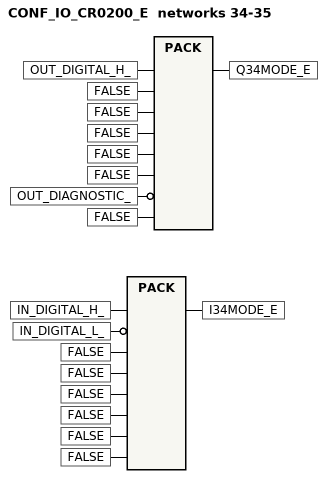
[picture p48: CONF_IO_CR0200_E (FBD) networks 34-35]
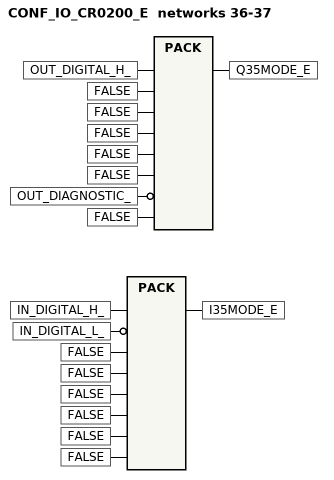
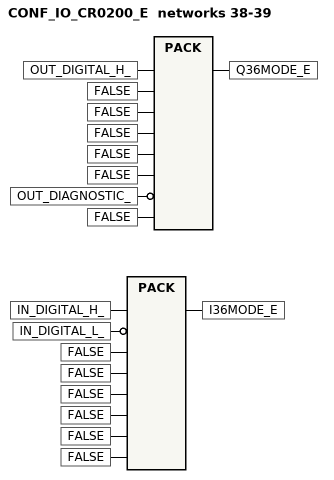
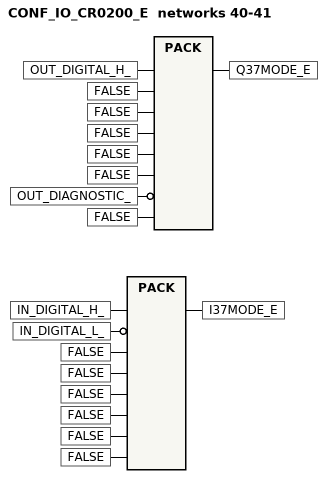
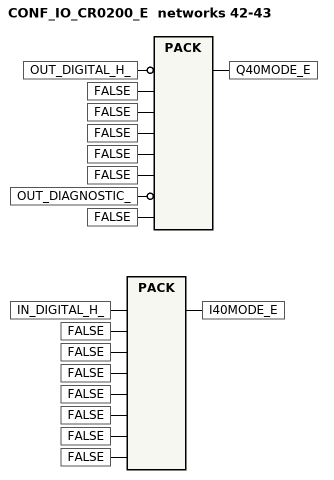
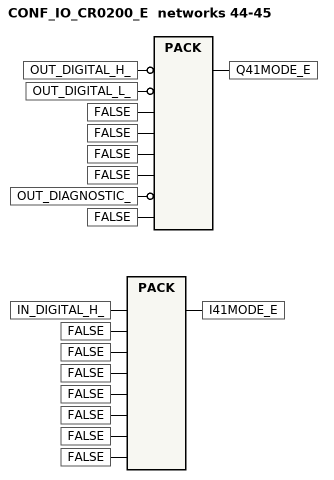
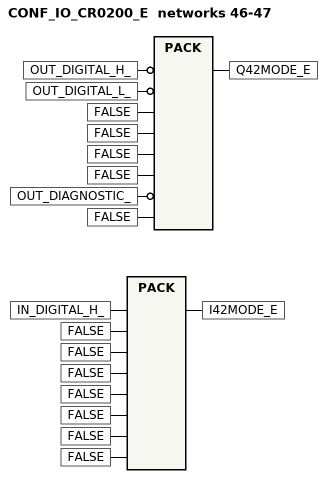
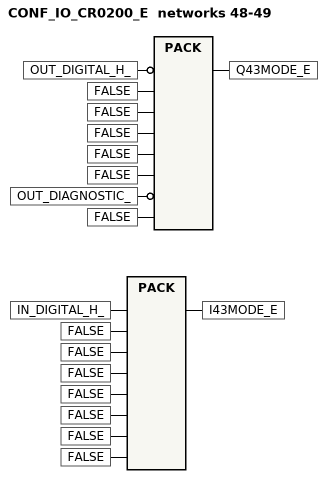
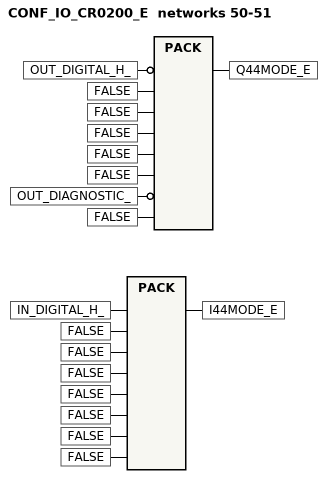
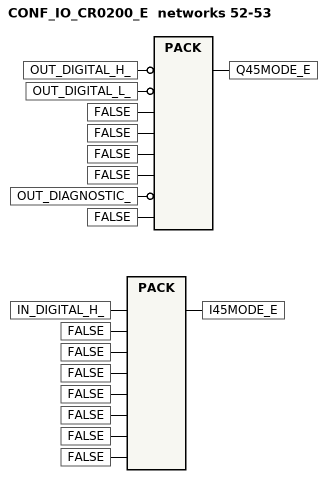
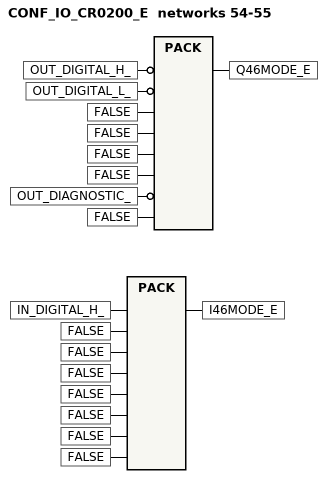
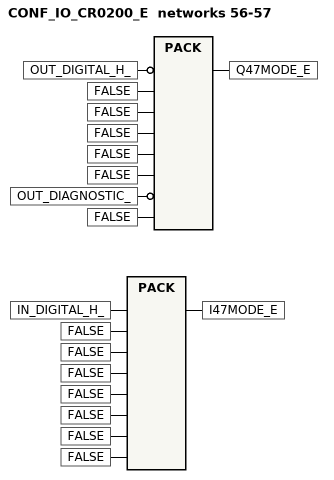
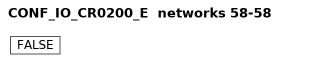
_FBD_ (* Function Block Diagram *)
NETWORK 1
	NOT init => >>END
NETWORK 2 (* Configuration byte for analog channel 0 pin 08 Connector 2. No output is connected to this pin. / Default setting:B0:=TRUE,B1:= FALSE,B2:= FALSE,B3:= FALSE,B4:= TRUE,B5:= FALSE,B6:= FALSE,B7:=FALSE *)
	PACK(IN_DIGITAL_H_, FALSE, NOT IN_CURRENT_, NOT IN_VOLTAGE10_, IN_VOLTAGE30_, NOT IN_RATIO_, FALSE, FALSE) => I00MODE_E
NETWORK 3 (* Configuration byte for analog channel 1 pin 27 Connector 2. No output is connected to this pin. / Default setting:B0:=TRUE,B1:= FALSE,B2:= FALSE,B3:= FALSE,B4:= TRUE,B5:= FALSE,B6:= FALSE,B7:=FALSE *)
	PACK(IN_DIGITAL_H_, FALSE, NOT IN_CURRENT_, NOT IN_VOLTAGE10_, IN_VOLTAGE30_, NOT IN_RATIO_, FALSE, FALSE) => I01MODE_E
NETWORK 4 (* Configuration byte for analog channel 2 pin 09 Connector 2. No output is connected to this pin. / Default setting:B0:=TRUE,B1:= FALSE,B2:= FALSE,B3:= FALSE,B4:= TRUE,B5:= FALSE,B6:= FALSE,B7:=FALSE *)
	PACK(IN_DIGITAL_H_, FALSE, NOT IN_CURRENT_, NOT IN_VOLTAGE10_, IN_VOLTAGE30_, NOT IN_RATIO_, FALSE, FALSE) => I02MODE_E
NETWORK 5 (* Configuration byte for analog channel 3 pin 28 Connector 2. No output is connected to this pin. / Default setting:B0:=TRUE,B1:= FALSE,B2:= FALSE,B3:= FALSE,B4:= TRUE,B5:= FALSE,B6:= FALSE,B7:=FALSE *)
	PACK(IN_DIGITAL_H_, FALSE, NOT IN_CURRENT_, NOT IN_VOLTAGE10_, IN_VOLTAGE30_, NOT IN_RATIO_, FALSE, FALSE) => I03MODE_E
NETWORK 6 (* Configuration byte for analog channel 4 pin 10 Connector 2. No output is connected to this pin. / Default setting:B0:=TRUE,B1:= FALSE,B2:= FALSE,B3:= FALSE,B4:= TRUE,B5:= FALSE,B6:= FALSE,B7:=FALSE *)
	PACK(IN_DIGITAL_H_, FALSE, NOT IN_CURRENT_, NOT IN_VOLTAGE10_, IN_VOLTAGE30_, NOT IN_RATIO_, FALSE, FALSE) => I04MODE_E
NETWORK 7 (* Configuration byte for analog channel 5 pin 29 Connector 2. No output is connected to this pin. / Default setting:B0:=TRUE,B1:= FALSE,B2:= FALSE,B3:= FALSE,B4:= TRUE,B5:= FALSE,B6:= FALSE,B7:=FALSE *)
	PACK(IN_DIGITAL_H_, FALSE, NOT IN_CURRENT_, NOT IN_VOLTAGE10_, IN_VOLTAGE30_, NOT IN_RATIO_, FALSE, FALSE) => I05MODE_E
NETWORK 8 (* Configuration byte for analog channel 6 pin 11 Connector 2. No output is connected to this pin. / Default setting:B0:=TRUE,B1:= FALSE,B2:= FALSE,B3:= FALSE,B4:= TRUE,B5:= FALSE,B6:= FALSE,B7:=FALSE *)
	PACK(IN_DIGITAL_H_, FALSE, NOT IN_CURRENT_, NOT IN_VOLTAGE10_, IN_VOLTAGE30_, NOT IN_RATIO_, FALSE, FALSE) => I06MODE_E
NETWORK 9 (* Configuration byte for analog channel 7 pin 30 Connector 2. No output is connected to this pin. / Default setting:B0:=TRUE,B1:= FALSE,B2:= FALSE,B3:= FALSE,B4:= TRUE,B5:= FALSE,B6:= FALSE,B7:=FALSE *)
	PACK(IN_DIGITAL_H_, FALSE, NOT IN_CURRENT_, NOT IN_VOLTAGE10_, IN_VOLTAGE30_, NOT IN_RATIO_, FALSE, FALSE) => I07MODE_E
NETWORK 10 (* Configuration byte for input %IX32.12  pin 20 Connector 2. No output is connected to this pin. / Default setting:B0:=TRUE,B1:= FALSE,B2:= FALSE,B3:= FALSE,B4:= FALSE,B5:= FALSE,B6:= FALSE,B7:=FALSE *)
	PACK(IN_DIGITAL_H_, FALSE, FALSE, FALSE, FALSE, FALSE, FALSE, NOT IN_FAST_) => I14MODE_E
NETWORK 11 (* Configuration byte for input %IX32.13  pin 02 Connector 2. No output is connected to this pin. / Default setting:B0:=TRUE,B1:= FALSE,B2:= FALSE,B3:= FALSE,B4:= FALSE,B5:= FALSE,B6:= FALSE,B7:=FALSE *)
	PACK(IN_DIGITAL_H_, FALSE, FALSE, FALSE, FALSE, FALSE, FALSE, NOT IN_FAST_) => I15MODE_E
NETWORK 12 (* Configuration byte for input %IX32.14  pin 21 Connector 2. No output is connected to this pin. / Default setting:B0:=TRUE,B1:= FALSE,B2:= FALSE,B3:= FALSE,B4:= FALSE,B5:= FALSE,B6:= FALSE,B7:=FALSE *)
	PACK(IN_DIGITAL_H_, FALSE, FALSE, FALSE, FALSE, FALSE, FALSE, NOT IN_FAST_) => I16MODE_E
NETWORK 13 (* Configuration byte for input %IX32.15  pin 38 Connector 2. No output is connected to this pin. / Default setting:B0:=TRUE,B1:= FALSE,B2:= FALSE,B3:= FALSE,B4:= FALSE,B5:= FALSE,B6:= FALSE,B7:=FALSE *)
	PACK(IN_DIGITAL_H_, FALSE, FALSE, FALSE, FALSE, FALSE, FALSE, NOT IN_FAST_) => I17MODE_E
NETWORK 14 (* Configuration byte for input %IX33.04  pin 19 Connector 2. No output is connected to this pin. / Default setting:B0:=TRUE,B1:= FALSE,B2:= FALSE,B3:= FALSE,B4:= FALSE,B5:= FALSE,B6:= FALSE,B7:=FALSE *)
	PACK(IN_DIGITAL_H_, FALSE, FALSE, FALSE, FALSE, FALSE, FALSE, NOT IN_FAST_) => I24MODE_E
NETWORK 15 (* Configuration byte for input %IX33.05  pin 55 Connector 2. No output is connected to this pin. / Default setting:B0:=TRUE,B1:= FALSE,B2:= FALSE,B3:= FALSE,B4:= FALSE,B5:= FALSE,B6:= FALSE,B7:=FALSE *)
	PACK(IN_DIGITAL_H_, FALSE, FALSE, FALSE, FALSE, FALSE, FALSE, NOT IN_FAST_) => I25MODE_E
NETWORK 16 (* Configuration byte for input %IX33.06  pin 18 Connector 2. No output is connected to this pin. / Default setting:B0:=TRUE,B1:= FALSE,B2:= FALSE,B3:= FALSE,B4:= FALSE,B5:= FALSE,B6:= FALSE,B7:=FALSE *)
	PACK(IN_DIGITAL_H_, FALSE, FALSE, FALSE, FALSE, FALSE, FALSE, NOT IN_FAST_) => I26MODE_E
NETWORK 17 (* Configuration byte for input %IX33.07  pin 37 Connector 2. No output is connected to this pin. / Default setting:B0:=TRUE,B1:= FALSE,B2:= FALSE,B3:= FALSE,B4:= FALSE,B5:= FALSE,B6:= FALSE,B7:=FALSE *)
	PACK(IN_DIGITAL_H_, FALSE, FALSE, FALSE, FALSE, FALSE, FALSE, NOT IN_FAST_) => I27MODE_E
NETWORK 18 (* Configuration byte for output %QX32.00  pin 44 Connector 2. The input %IX32.08 on pin 44 has no configuration byte. / Default setting:B0:=TRUE,B1:= FALSE,B2:= FALSE,B3:= FALSE,B4:= FALSE,B5:= FALSE,B6:= FALSE,B7:=TRUE *)
	PACK(OUT_DIGITAL_H_, FALSE, NOT OUT_CURRENT_, FALSE, FALSE, FALSE, NOT OUT_DIAGNOSTIC_, OUT_OVERLOAD_PROTECTION_) => Q10MODE_E
NETWORK 19 (* Configuration byte for output %QX32.01  pin 45 Connector 2. The input %IX32.09 on pin 45 has no configuration byte. / Default setting:B0:=TRUE,B1:= FALSE,B2:= FALSE,B3:= FALSE,B4:= FALSE,B5:= FALSE,B6:= FALSE,B7:=TRUE *)
	PACK(OUT_DIGITAL_H_, FALSE, NOT OUT_CURRENT_, FALSE, FALSE, FALSE, NOT OUT_DIAGNOSTIC_, OUT_OVERLOAD_PROTECTION_) => Q11MODE_E
NETWORK 20 (* Configuration byte for output %QX32.02  pin 46 Connector 2. The input %IX32.10 on pin 46 has no configuration byte. / Default setting:B0:=TRUE,B1:= FALSE,B2:= FALSE,B3:= FALSE,B4:= FALSE,B5:= FALSE,B6:= FALSE,B7:=TRUE *)
	PACK(OUT_DIGITAL_H_, FALSE, NOT OUT_CURRENT_, FALSE, FALSE, FALSE, NOT OUT_DIAGNOSTIC_, OUT_OVERLOAD_PROTECTION_) => Q12MODE_E
NETWORK 21 (* Configuration byte for output %QX32.03  pin 47 Connector 2. The input %IX32.11 on pin 47 has no configuration byte. / Default setting:B0:=TRUE,B1:= FALSE,B2:= FALSE,B3:= FALSE,B4:= FALSE,B5:= FALSE,B6:= FALSE,B7:=TRUE *)
	PACK(OUT_DIGITAL_H_, FALSE, NOT OUT_CURRENT_, FALSE, FALSE, FALSE, NOT OUT_DIAGNOSTIC_, OUT_OVERLOAD_PROTECTION_) => Q13MODE_E
NETWORK 22 (* Configuration byte for output %QX32.04  pin 36 Connector 2. The input %IX33.00 on pin 36 has no configuration byte. / Default setting:B0:=TRUE,B1:= FALSE,B2:= FALSE,B3:= FALSE,B4:= FALSE,B5:= FALSE,B6:= FALSE,B7:=TRUE *)
	PACK(OUT_DIGITAL_H_, FALSE, NOT OUT_CURRENT_, FALSE, FALSE, FALSE, NOT OUT_DIAGNOSTIC_, OUT_OVERLOAD_PROTECTION_) => Q20MODE_E
NETWORK 23 (* Configuration byte for output %QX32.05  pin 54 Connector 2 The input %IX33.01 on pin 54 has no configuration byte. / Default setting:B0:=TRUE,B1:= FALSE,B2:= FALSE,B3:= FALSE,B4:= FALSE,B5:= FALSE,B6:= FALSE,B7:=TRUE *)
	PACK(OUT_DIGITAL_H_, FALSE, NOT OUT_CURRENT_, FALSE, FALSE, FALSE, NOT OUT_DIAGNOSTIC_, OUT_OVERLOAD_PROTECTION_) => Q21MODE_E
NETWORK 24 (* Configuration byte for output %QX32.06  pin 17 Connector 2 The input %IX33.02 on pin 17 has no configuration byte. / Default setting:B0:=TRUE,B1:= FALSE,B2:= FALSE,B3:= FALSE,B4:= FALSE,B5:= FALSE,B6:= FALSE,B7:=TRUE *)
	PACK(OUT_DIGITAL_H_, FALSE, NOT OUT_CURRENT_, FALSE, FALSE, FALSE, NOT OUT_DIAGNOSTIC_, OUT_OVERLOAD_PROTECTION_) => Q22MODE_E
NETWORK 25 (* Configuration byte for output %QX32.07  pin 53 Connector 2 The input %IX33.03 on pin 53 has no configuration byte. / Default setting:B0:=TRUE,B1:= FALSE,B2:= FALSE,B3:= FALSE,B4:= FALSE,B5:= FALSE,B6:= FALSE,B7:=TRUE *)
	PACK(OUT_DIGITAL_H_, FALSE, NOT OUT_CURRENT_, FALSE, FALSE, FALSE, NOT OUT_DIAGNOSTIC_, OUT_OVERLOAD_PROTECTION_) => Q23MODE_E
NETWORK 26 (* Configuration byte for output %QX32.08  pin 39 Connector 2. / Default setting:B0:=TRUE,B1:= FALSE,B2:= FALSE,B3:= FALSE,B4:= FALSE,B5:= FALSE,B6:= FALSE,B7:=FALSE *)
	PACK(OUT_DIGITAL_H_, FALSE, FALSE, FALSE, FALSE, FALSE, NOT OUT_DIAGNOSTIC_, FALSE) => Q30MODE_E
NETWORK 27 (* Configuration byte for input %IX33.08  pin 39 Connector 2. / Default setting:B0:=TRUE,B1:= FALSE,B2:= FALSE,B3:= FALSE,B4:= FALSE,B5:= FALSE,B6:= FALSE,B7:=FALSE *)
	PACK(IN_DIGITAL_H_, NOT IN_DIGITAL_L_, FALSE, FALSE, FALSE, FALSE, FALSE, FALSE) => I30MODE_E
NETWORK 28 (* Configuration byte for output %QX32.09  pin 03 Connector 2. / Default setting:B0:=TRUE,B1:= FALSE,B2:= FALSE,B3:= FALSE,B4:= FALSE,B5:= FALSE,B6:= FALSE,B7:=FALSE *)
	PACK(OUT_DIGITAL_H_, FALSE, FALSE, FALSE, FALSE, FALSE, NOT OUT_DIAGNOSTIC_, FALSE) => Q31MODE_E
NETWORK 29 (* Configuration byte for input %IX33.09  pin 03 Connector 2. / Default setting:B0:=TRUE,B1:= FALSE,B2:= FALSE,B3:= FALSE,B4:= FALSE,B5:= FALSE,B6:= FALSE,B7:=FALSE *)
	PACK(IN_DIGITAL_H_, NOT IN_DIGITAL_L_, FALSE, FALSE, FALSE, FALSE, FALSE, FALSE) => I31MODE_E
NETWORK 30 (* Configuration byte for output %QX32.10  pin 40 Connector 2. / Default setting:B0:=TRUE,B1:= FALSE,B2:= FALSE,B3:= FALSE,B4:= FALSE,B5:= FALSE,B6:= FALSE,B7:=FALSE *)
	PACK(OUT_DIGITAL_H_, FALSE, FALSE, FALSE, FALSE, FALSE, NOT OUT_DIAGNOSTIC_, FALSE) => Q32MODE_E
NETWORK 31 (* Configuration byte forintput %IX33.10  pin 40 Connector 2. / Default setting:B0:=TRUE,B1:= FALSE,B2:= FALSE,B3:= FALSE,B4:= FALSE,B5:= FALSE,B6:= FALSE,B7:=FALSE *)
	PACK(IN_DIGITAL_H_, NOT IN_DIGITAL_L_, FALSE, FALSE, FALSE, FALSE, FALSE, FALSE) => I32MODE_E
NETWORK 32 (* Configuration byte for output %QX32.11  pin 22 Connector 2. / Default setting:B0:=TRUE,B1:= FALSE,B2:= FALSE,B3:= FALSE,B4:= FALSE,B5:= FALSE,B6:= FALSE,B7:=FALSE *)
	PACK(OUT_DIGITAL_H_, FALSE, FALSE, FALSE, FALSE, FALSE, NOT OUT_DIAGNOSTIC_, FALSE) => Q33MODE_E
NETWORK 33 (* Configuration byte for input %IX33.11  pin 22 Connector 2. / Default setting:B0:=TRUE,B1:= FALSE,B2:= FALSE,B3:= FALSE,B4:= FALSE,B5:= FALSE,B6:= FALSE,B7:=FALSE *)
	PACK(IN_DIGITAL_H_, NOT IN_DIGITAL_L_, FALSE, FALSE, FALSE, FALSE, FALSE, FALSE) => I33MODE_E
NETWORK 34 (* Configuration byte for output %QX32.12  pin 41 Connector 2. / Default setting:B0:=TRUE,B1:= FALSE,B2:= FALSE,B3:= FALSE,B4:= FALSE,B5:= FALSE,B6:= FALSE,B7:=FALSE *)
	PACK(OUT_DIGITAL_H_, FALSE, FALSE, FALSE, FALSE, FALSE, NOT OUT_DIAGNOSTIC_, FALSE) => Q34MODE_E
NETWORK 35 (* Configuration byte for input %IX33.12  pin 41 Connector 2. / Default setting:B0:=TRUE,B1:= FALSE,B2:= FALSE,B3:= FALSE,B4:= FALSE,B5:= FALSE,B6:= FALSE,B7:=FALSE *)
	PACK(IN_DIGITAL_H_, NOT IN_DIGITAL_L_, FALSE, FALSE, FALSE, FALSE, FALSE, FALSE) => I34MODE_E
NETWORK 36 (* Configuration byte for output %QX32.13  pin 42 Connector 2. / Default setting:B0:=TRUE,B1:= FALSE,B2:= FALSE,B3:= FALSE,B4:= FALSE,B5:= FALSE,B6:= FALSE,B7:=FALSE *)
	PACK(OUT_DIGITAL_H_, FALSE, FALSE, FALSE, FALSE, FALSE, NOT OUT_DIAGNOSTIC_, FALSE) => Q35MODE_E
NETWORK 37 (* Configuration byte for input %IX33.13  pin 42 Connector 2. / Default setting:B0:=TRUE,B1:= FALSE,B2:= FALSE,B3:= FALSE,B4:= FALSE,B5:= FALSE,B6:= FALSE,B7:=FALSE *)
	PACK(IN_DIGITAL_H_, NOT IN_DIGITAL_L_, FALSE, FALSE, FALSE, FALSE, FALSE, FALSE) => I35MODE_E
NETWORK 38 (* Configuration byte for output %QX32.14  pin 43 Connector 2. / Default setting:B0:=TRUE,B1:= FALSE,B2:= FALSE,B3:= FALSE,B4:= FALSE,B5:= FALSE,B6:= FALSE,B7:=FALSE *)
	PACK(OUT_DIGITAL_H_, FALSE, FALSE, FALSE, FALSE, FALSE, NOT OUT_DIAGNOSTIC_, FALSE) => Q36MODE_E
NETWORK 39 (* Configuration byte for input %IX33.14  pin 43 Connector 2. / Default setting:B0:=TRUE,B1:= FALSE,B2:= FALSE,B3:= FALSE,B4:= FALSE,B5:= FALSE,B6:= FALSE,B7:=FALSE *)
	PACK(IN_DIGITAL_H_, NOT IN_DIGITAL_L_, FALSE, FALSE, FALSE, FALSE, FALSE, FALSE) => I36MODE_E
NETWORK 40 (* Configuration byte for output %QX32.15  pin 04 Connector 2. / Default setting:B0:=TRUE,B1:= FALSE,B2:= FALSE,B3:= FALSE,B4:= FALSE,B5:= FALSE,B6:= FALSE,B7:=FALSE *)
	PACK(OUT_DIGITAL_H_, FALSE, FALSE, FALSE, FALSE, FALSE, NOT OUT_DIAGNOSTIC_, FALSE) => Q37MODE_E
NETWORK 41 (* Configuration byte for input %IX33.15  pin 04 Connector 2. / Default setting:B0:=TRUE,B1:= FALSE,B2:= FALSE,B3:= FALSE,B4:= FALSE,B5:= FALSE,B6:= FALSE,B7:=FALSE *)
	PACK(IN_DIGITAL_H_, NOT IN_DIGITAL_L_, FALSE, FALSE, FALSE, FALSE, FALSE, FALSE) => I37MODE_E
NETWORK 42 (* Configuration byte for output %QX33.00  pin 48 Connector 2. / Default setting:B0:=FALSE,B1:= FALSE,B2:= FALSE,B3:= FALSE,B4:= FALSE,B5:= FALSE,B6:= FALSE,B7:=FALSE *)
	PACK(NOT OUT_DIGITAL_H_, FALSE, FALSE, FALSE, FALSE, FALSE, NOT OUT_DIAGNOSTIC_, FALSE) => Q40MODE_E
NETWORK 43 (* Configuration byte for intput %IX34.00  pin 48 Connector 2. / Default setting:B0:=TRUE,B1:= FALSE,B2:= FALSE,B3:= FALSE,B4:= FALSE,B5:= FALSE,B6:= FALSE,B7:=FALSE *)
	PACK(IN_DIGITAL_H_, FALSE, FALSE, FALSE, FALSE, FALSE, FALSE, FALSE) => I40MODE_E
NETWORK 44 (* Configuration byte for output %QX33.01  pin 49 Connector 2. / Default setting:B0:=FALSE,B1:= FALSE,B2:= FALSE,B3:= FALSE,B4:= FALSE,B5:= FALSE,B6:= FALSE,B7:=FALSE *)
	PACK(NOT OUT_DIGITAL_H_, NOT OUT_DIGITAL_L_, FALSE, FALSE, FALSE, FALSE, NOT OUT_DIAGNOSTIC_, FALSE) => Q41MODE_E
NETWORK 45 (* Configuration byte for input %IX34.01  pin 49 Connector 2. / Default setting:B0:=TRUE,B1:= FALSE,B2:= FALSE,B3:= FALSE,B4:= FALSE,B5:= FALSE,B6:= FALSE,B7:=FALSE *)
	PACK(IN_DIGITAL_H_, FALSE, FALSE, FALSE, FALSE, FALSE, FALSE, FALSE) => I41MODE_E
NETWORK 46 (* Configuration byte for output %QX33.02  pin 31 Connector 2. / Default setting:B0:=FALSE,B1:= FALSE,B2:= FALSE,B3:= FALSE,B4:= FALSE,B5:= FALSE,B6:= FALSE,B7:=FALSE *)
	PACK(NOT OUT_DIGITAL_H_, NOT OUT_DIGITAL_L_, FALSE, FALSE, FALSE, FALSE, NOT OUT_DIAGNOSTIC_, FALSE) => Q42MODE_E
NETWORK 47 (* Configuration byte for input %IX34.02  pin 31 Connector 2. / Default setting:B0:=TRUE,B1:= FALSE,B2:= FALSE,B3:= FALSE,B4:= FALSE,B5:= FALSE,B6:= FALSE,B7:=FALSE *)
	PACK(IN_DIGITAL_H_, FALSE, FALSE, FALSE, FALSE, FALSE, FALSE, FALSE) => I42MODE_E
NETWORK 48 (* Configuration byte for output %QX33.03  pin 50 Connector 2. / Default setting:B0:=FALSE,B1:= FALSE,B2:= FALSE,B3:= FALSE,B4:= FALSE,B5:= FALSE,B6:= FALSE,B7:=FALSE *)
	PACK(NOT OUT_DIGITAL_H_, FALSE, FALSE, FALSE, FALSE, FALSE, NOT OUT_DIAGNOSTIC_, FALSE) => Q43MODE_E
NETWORK 49 (* Configuration byte for input %IX34.03  pin 50 Connector 2. / Default setting:B0:=TRUE,B1:= FALSE,B2:= FALSE,B3:= FALSE,B4:= FALSE,B5:= FALSE,B6:= FALSE,B7:=FALSE *)
	PACK(IN_DIGITAL_H_, FALSE, FALSE, FALSE, FALSE, FALSE, FALSE, FALSE) => I43MODE_E
NETWORK 50 (* Configuration byte for output %QX33.04  pin 51 Connector 2. / Default setting:B0:=FALSE,B1:= FALSE,B2:= FALSE,B3:= FALSE,B4:= FALSE,B5:= FALSE,B6:= FALSE,B7:=FALSE *)
	PACK(NOT OUT_DIGITAL_H_, FALSE, FALSE, FALSE, FALSE, FALSE, NOT OUT_DIAGNOSTIC_, FALSE) => Q44MODE_E
NETWORK 51 (* Configuration byte for input %IX34.04  pin 51 Connector 2. / Default setting:B0:=TRUE,B1:= FALSE,B2:= FALSE,B3:= FALSE,B4:= FALSE,B5:= FALSE,B6:= FALSE,B7:=FALSE *)
	PACK(IN_DIGITAL_H_, FALSE, FALSE, FALSE, FALSE, FALSE, FALSE, FALSE) => I44MODE_E
NETWORK 52 (* Configuration byte for output %QX33.05  pin 52 Connector 2. / Default setting:B0:=FALSE,B1:= FALSE,B2:= FALSE,B3:= FALSE,B4:= FALSE,B5:= FALSE,B6:= FALSE,B7:=FALSE *)
	PACK(NOT OUT_DIGITAL_H_, NOT OUT_DIGITAL_L_, FALSE, FALSE, FALSE, FALSE, NOT OUT_DIAGNOSTIC_, FALSE) => Q45MODE_E
NETWORK 53 (* Configuration byte for input %IX33.05  pin 52 Connector 2. / Default setting:B0:=TRUE,B1:= FALSE,B2:= FALSE,B3:= FALSE,B4:= FALSE,B5:= FALSE,B6:= FALSE,B7:=FALSE *)
	PACK(IN_DIGITAL_H_, FALSE, FALSE, FALSE, FALSE, FALSE, FALSE, FALSE) => I45MODE_E
NETWORK 54 (* Configuration byte for output %QX33.06  pin 16 Connector 2. / Default setting:B0:=FALSE,B1:= FALSE,B2:= FALSE,B3:= FALSE,B4:= FALSE,B5:= FALSE,B6:= FALSE,B7:=FALSE *)
	PACK(NOT OUT_DIGITAL_H_, NOT OUT_DIGITAL_L_, FALSE, FALSE, FALSE, FALSE, NOT OUT_DIAGNOSTIC_, FALSE) => Q46MODE_E
NETWORK 55 (* Configuration byte for input %IX34.06  pin 16 Connector 2. / Default setting:B0:=TRUE,B1:= FALSE,B2:= FALSE,B3:= FALSE,B4:= FALSE,B5:= FALSE,B6:= FALSE,B7:=FALSE *)
	PACK(IN_DIGITAL_H_, FALSE, FALSE, FALSE, FALSE, FALSE, FALSE, FALSE) => I46MODE_E
NETWORK 56 (* Configuration byte for output %QX33.07  pin 35 Connector 2. / Default setting:B0:=FALSE,B1:= FALSE,B2:= FALSE,B3:= FALSE,B4:= FALSE,B5:= FALSE,B6:= FALSE,B7:=FALSE *)
	PACK(NOT OUT_DIGITAL_H_, FALSE, FALSE, FALSE, FALSE, FALSE, NOT OUT_DIAGNOSTIC_, FALSE) => Q47MODE_E
NETWORK 57 (* Configuration byte for input %IX34.07  pin 35 Connector 2. / Default setting:B0:=TRUE,B1:= FALSE,B2:= FALSE,B3:= FALSE,B4:= FALSE,B5:= FALSE,B6:= FALSE,B7:=FALSE *)
	PACK(IN_DIGITAL_H_, FALSE, FALSE, FALSE, FALSE, FALSE, FALSE, FALSE) => I47MODE_E
NETWORK 58 END::
	FALSE
_END_FBD_
END_PROGRAM

(* POU POUS, ST *)
PROGRAM POUS
VAR

END_VAR
	mv_alarm10001			:=0;
	mv_alarm10002			:=0;
	mv_alarm10003			:=0;
	mv_alarm10004			:=0;
	mv_alarm10005 			:=0;
	mv_alarm10006 			:=0;
	mv_alarm10007 			:=0;
	mv_alarm10008			:=0;
	mv_alarm10009			:=0;
	mv_alarm10010			:=0;
	mv_alarm10011			:=0;
	mv_alarm10012			:=0;
	mv_alarm10013			:=0;
	mv_alarm10014 			:=0;
	mv_alarm10015 			:=0;
	mv_alarm10016 			:=0;


	IO_CONFIG();
	SPEED_ASSIGN();
	LEVEL();
	DOWN_PART_DEAL();
	COM_ERROR();
	DATA_ACTIONG();
	ALARM_TEXT();
END_PROGRAM

(* POU I_O_CONFIGURATION/VEHICLE/IO_CONFIG, ST *)
PROGRAM IO_CONFIG
VAR
END_VAR
CASE vehicle_styel OF
10011:
	io_config_address_10011();
	io_config_10011();
10012:
	io_config_address_10012();
	io_config_10012();
10013:
	io_config_address_10013();
	io_config_10013();
10014:
	io_config_address_10014();
	io_config_10014();
ELSE
	io_config_address_10013();
	io_config_10013();
END_CASE
END_PROGRAM

(* POU I_O_CONFIGURATION/VEHICLE/io_config_address_10011, ST *)
PROGRAM io_config_address_10011
VAR
END_VAR
	front_left_Lv_ex_check1		:= %IX0.6			;	(*左前水平伸到位*)
	front_right_Lv_ex_check1		:= %IX0.7			;	(*右前水平伸到位*)
	back_left_Lv_ex_check1		:= %IX0.12			;	(*左后水平伸到位*)
	back_right_Lv_ex_check1	:= %IX0.13			;	(*右后水平伸到位*)
	front_left_urt_ex_check1		:= %IX0.14			;	(*左前垂直伸到位*)
	front_right_urt_ex_check1	:= %IX0.15			;	(*右前垂直伸到位*)
	back_left_urt_ex_check1		:= %IX1.4			;	(*左后垂直伸到位*)
	back_right_urt_ex_check1	:= %IX1.5			;	(*右后垂直伸到位*)

	front_left_Lv_drb_check		:= %IX32.1			;	(*左前水平收到位*)
	front_right_Lv_drb_check		:= %IX32.2			;	(*右前水平收到位*)
	back_left_Lv_drb_check		:= %IX32.3			;	(*左后水平收到位*)
	back_right_Lv_drb_check	:= %IX32.4			;	(*右后水平收到位*)
	front_left_urt_drb_check1		:= %IX32.5			;	(*左前垂直收到位*)
	front_right_urt_drb_check1	:= %IX32.6			;	(*右前垂直收到位*)
	back_left_urt_drb_check1	:= %IX32.7			;	(*左后垂直收到位*)
	back_right_urt_drb_check1	:= %IX32.12		;	(*右后垂直收到位*)

	engine_run					:= %IX2.2			;	(*发动机启动*)
	engine_stop					:= %IX2.3			;	(*发动机停止*)
	accelerate_sb					:= %IX2.0			;	(*加速*)
	decelerate_sb					:= %IX2.1			;	(*减速*)

(***操作***)
	tt_forcexx						:= %IX34.6			;	(*转台强制*)
	down_force					:= %IX34.7			;	(*下车强制*)
	auto_manu_choice			:= %IX34.1			;	(*自动/手动*)
	water_pump_run_sb			:= %IX1.7			;	(*消防泵开*)

	level_extend_triger_left1		:= %IX34.2			;	(*自动伸支腿*)
	level_extend_triger_right1	:= %IX34.3			;	(*自动伸支腿*)
	auto_extend_triger_left1		:= %IX33.5			;	(*自动伸支腿*)
	auto_extend_triger_right1	:= %IX33.6			;	(*自动伸支腿*)
	auto_drawback_triger_left1	:= %IX33.7			;	(*自动收支腿*)
	auto_drawback_triger_right1	:= %IX34.0			;	(*自动收支腿*)

	arm_to_station				:= %IX2.4			;	(*臂架到位检测*)
	water_pump_check			:= %IX33.4			;	(*水泵取力*)
	left_groud_check1			:= %IX34.4			;	(*车胎离地1*)
	left_groud_check2			:= %IX34.5			;	(*车胎离地2*)

	%QX32.2						:=	left_front_lv_ex_valve					;	(*左前水平伸*)
 	%QX32.0 						:=	left_back_lv_ex_valve					;	(*左后水平伸*)
 	%QX32.6						:=	right_front_lv_ex_valve				;	(*右前水平伸*)
	%QX32.4						:=	right_back_lv_ex_valve				;	(*右后水平伸*)
	%QX32.3						:=	left_front_lv_drb_valve				;	(*左前水平收*)
	%QX32.1						:=	left_back_lv_drb_valve				;	(*左后水平收*)
	%QX32.7						:=	right_front_lv_drb_valve				;	(*右前水平收*)
 	%QX32.5						:=	right_back_lv_drb_valve				;	(*右后水平收*)

(***底盘***)
	%QX0.8						:=	enginer_run_ctl						;	(*启动控制*)
	%QX0.9						:=	enginer_stop_ctl						;	(*熄火控制*)
 	%QX32.9						:=	enginer_acc_ctl						;	(*加速控制*)
	%QX32.10						:=	enginer_dec_ctl						;	(*减速控制*)

(***操作***)
	%QX0.10						:=	water_pump_ctl						;	(*水泵控制*)
	%QX32.14						:=	up_valve_ctl							;	(*上车阀*)
	%QX32.15						:=	down_valve_ctl						;	(*下车阀*)

(***指示***)
	%QX0.11						:=	over_level_sign						;	(*坡度超限*)
	%QX0.12						:=	triger_left_grd_sign					;	(*支腿离地*)
	%QX32.8						:=	alarmer_horn							;	(*警报器*)
	%QX32.13						:=	triger_flash							;	(*支腿闪光灯*)
	%QX0.10						:=	water_pump_ctl_sign					;	(*水泵控制指示*)

	%QX0.14						:=	left_f_lv_ex_over						;	(*左前水平伸到位*)
	%QX0.15						:=	left_b_lv_ex_over						;	(*左后水平伸到位*)
	%QX32.11						:=	right_f_lv_ex_over						;	(*右前水平伸到位*)
	%QX32.12						:=	right_b_lv_ex_over					;	(*右后水平伸到位*)
END_PROGRAM

(* POU I_O_CONFIGURATION/VEHICLE/io_config_10011, FBD *)
PROGRAM io_config_10011
VAR
	CH_NO1: INPUT_ANALOG;
	CH_NO2: INPUT_ANALOG;
	CH_NO3: INPUT_ANALOG;
	CH_NO4: INPUT_ANALOG;
	CH_NO5: INPUT_ANALOG_E;
	CH_NO6: FREQUENCY_E;



END_VAR
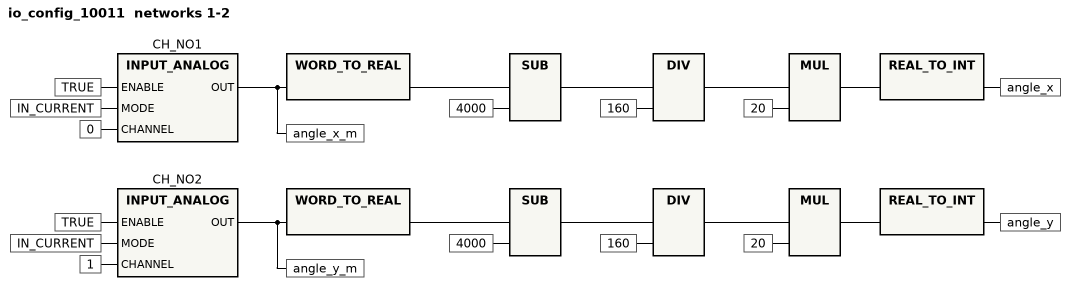
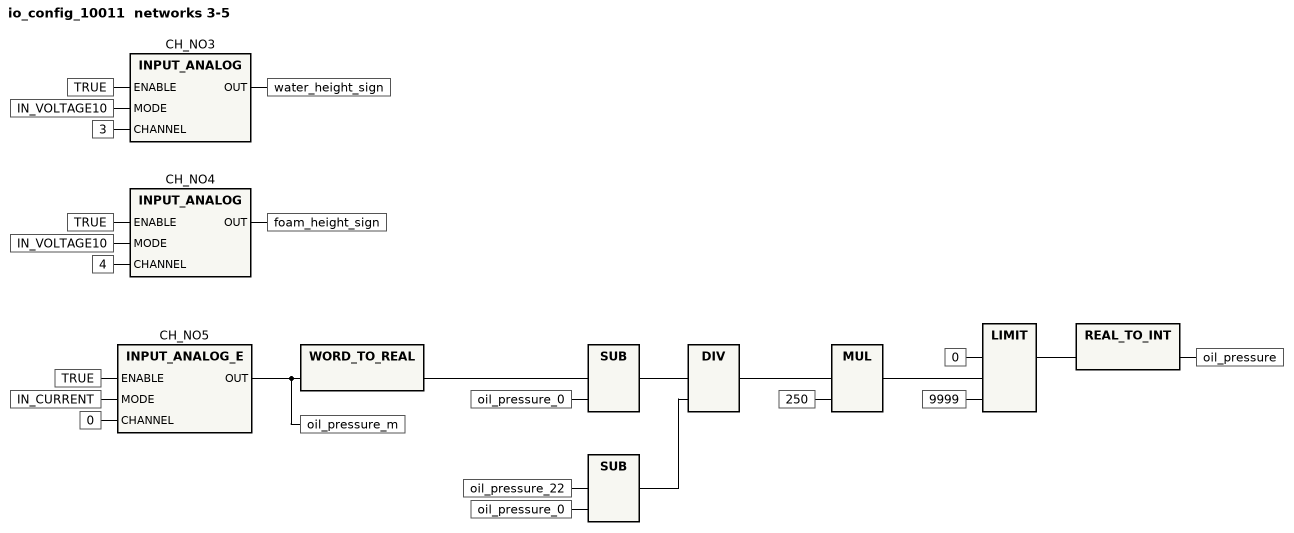
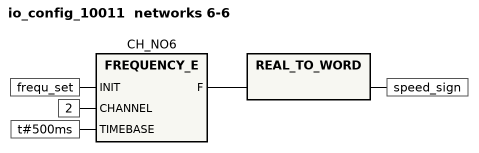
_FBD_ (* Function Block Diagram *)
NETWORK 1
	REAL_TO_INT(MUL(DIV(SUB(WORD_TO_REAL(<CH_NO1:INPUT_ANALOG(ENABLE: TRUE, MODE: IN_CURRENT, CHANNEL: 0) => angle_x_m>), 4000), 160), 20)) => angle_x
NETWORK 2
	REAL_TO_INT(MUL(DIV(SUB(WORD_TO_REAL(<CH_NO2:INPUT_ANALOG(ENABLE: TRUE, MODE: IN_CURRENT, CHANNEL: 1) => angle_y_m>), 4000), 160), 20)) => angle_y
NETWORK 3
	CH_NO3:INPUT_ANALOG(ENABLE: TRUE, MODE: IN_VOLTAGE10, CHANNEL: 3) => water_height_sign
NETWORK 4
	CH_NO4:INPUT_ANALOG(ENABLE: TRUE, MODE: IN_VOLTAGE10, CHANNEL: 4) => foam_height_sign
NETWORK 5
	REAL_TO_INT(LIMIT(0, MUL(DIV(SUB(WORD_TO_REAL(<CH_NO5:INPUT_ANALOG_E(ENABLE: TRUE, MODE: IN_CURRENT, CHANNEL: 0) => oil_pressure_m>), oil_pressure_0), SUB(oil_pressure_22, oil_pressure_0)), 250), 9999)) => oil_pressure
NETWORK 6
	REAL_TO_WORD(CH_NO6:FREQUENCY_E(INIT: frequ_set, CHANNEL: 2, TIMEBASE: t#500ms)) => speed_sign
_END_FBD_
(* the same logic as Structured Text *)
(* Network 1 *)
CH_NO1(ENABLE := TRUE, MODE := IN_CURRENT, CHANNEL := 0);
angle_x_m := CH_NO1.OUT;
angle_x := REAL_TO_INT(((WORD_TO_REAL(CH_NO1.OUT) - 4000) / 160) * 20);
(* Network 2 *)
CH_NO2(ENABLE := TRUE, MODE := IN_CURRENT, CHANNEL := 1);
angle_y_m := CH_NO2.OUT;
angle_y := REAL_TO_INT(((WORD_TO_REAL(CH_NO2.OUT) - 4000) / 160) * 20);
(* Network 3 *)
CH_NO3(ENABLE := TRUE, MODE := IN_VOLTAGE10, CHANNEL := 3);
water_height_sign := CH_NO3.OUT;
(* Network 4 *)
CH_NO4(ENABLE := TRUE, MODE := IN_VOLTAGE10, CHANNEL := 4);
foam_height_sign := CH_NO4.OUT;
(* Network 5 *)
CH_NO5(ENABLE := TRUE, MODE := IN_CURRENT, CHANNEL := 0);
oil_pressure_m := CH_NO5.OUT;
oil_pressure := REAL_TO_INT(LIMIT(0, ((WORD_TO_REAL(CH_NO5.OUT) - oil_pressure_0) / (oil_pressure_22 - oil_pressure_0)) * 250, 9999));
(* Network 6 *)
CH_NO6(INIT := frequ_set, CHANNEL := 2, TIMEBASE := t#500ms);
speed_sign := REAL_TO_WORD(CH_NO6.F);
END_PROGRAM

(* POU I_O_CONFIGURATION/VEHICLE/io_config_address_10012, ST *)
PROGRAM io_config_address_10012
VAR
END_VAR
	front_left_Lv_ex_check1		:= %IX0.6			;	(*左前水平伸到位*)
	front_right_Lv_ex_check1		:= %IX0.7			;	(*右前水平伸到位*)
	back_left_Lv_ex_check1		:= %IX0.12			;	(*左后水平伸到位*)
	back_right_Lv_ex_check1	:= %IX0.13			;	(*右后水平伸到位*)
	front_left_urt_ex_check1		:= %IX0.14			;	(*左前垂直伸到位*)
	front_right_urt_ex_check1	:= %IX0.15			;	(*右前垂直伸到位*)
	back_left_urt_ex_check1		:= %IX1.4			;	(*左后垂直伸到位*)
	back_right_urt_ex_check1	:= %IX1.5			;	(*右后垂直伸到位*)

	front_left_Lv_drb_check		:= %IX32.1			;	(*左前水平收到位*)
	front_right_Lv_drb_check		:= %IX32.2			;	(*右前水平收到位*)
	back_left_Lv_drb_check		:= %IX32.3			;	(*左后水平收到位*)
	back_right_Lv_drb_check	:= %IX32.4			;	(*右后水平收到位*)
	front_left_urt_drb_check1		:= %IX32.5			;	(*左前垂直收到位*)
	front_right_urt_drb_check1	:= %IX32.6			;	(*右前垂直收到位*)
	back_left_urt_drb_check1	:= %IX32.7			;	(*左后垂直收到位*)
	back_right_urt_drb_check1	:= %IX32.12		;	(*右后垂直收到位*)

	engine_run					:= %IX2.2			;	(*发动机启动*)
	engine_stop					:= %IX2.3			;	(*发动机停止*)
	accelerate_sb					:= %IX2.0			;	(*加速*)
	decelerate_sb					:= %IX2.1			;	(*减速*)

(***操作***)
	tt_forcexx						:= %IX34.6			;	(*转台强制*)
	down_force					:= %IX34.7			;	(*下车强制*)
	auto_manu_choice			:= %IX34.1			;	(*自动/手动*)
	water_pump_run_sb			:= %IX1.7			;	(*消防泵开*)








	arm_to_station				:= %IX2.4			;	(*臂架到位检测*)
	water_pump_check			:= %IX33.4			;	(*水泵取力*)
	left_groud_check1			:= %IX34.4			;	(*车胎离地1*)
	left_groud_check2			:= %IX34.5			;	(*车胎离地2*)

	%QX32.2						:=	left_front_lv_ex_valve					;	(*左前水平伸*)
 	%QX32.0 						:=	left_back_lv_ex_valve					;	(*左后水平伸*)
 	%QX32.6						:=	right_front_lv_ex_valve				;	(*右前水平伸*)
	%QX32.4						:=	right_back_lv_ex_valve				;	(*右后水平伸*)
	%QX32.3						:=	left_front_lv_drb_valve				;	(*左前水平收*)
	%QX32.1						:=	left_back_lv_drb_valve				;	(*左后水平收*)
	%QX32.7						:=	right_front_lv_drb_valve				;	(*右前水平收*)
 	%QX32.5						:=	right_back_lv_drb_valve				;	(*右后水平收*)

(***底盘***)
	%QX0.8						:=	enginer_run_ctl						;	(*启动控制*)
	%QX0.9						:=	enginer_stop_ctl						;	(*熄火控制*)
 	%QX32.9						:=	enginer_acc_ctl						;	(*加速控制*)
	%QX32.10						:=	enginer_dec_ctl						;	(*减速控制*)

(***操作***)
	%QX0.10						:=	water_pump_ctl						;	(*水泵控制*)
	%QX32.14						:=	up_valve_ctl							;	(*上车阀*)
	%QX32.15						:=	down_valve_ctl						;	(*下车阀*)

(***指示***)
	%QX0.11						:=	over_level_sign						;	(*坡度超限*)
	%QX0.12						:=	triger_left_grd_sign					;	(*支腿离地*)
	%QX32.8						:=	alarmer_horn							;	(*警报器*)
	%QX32.13						:=	triger_flash							;	(*支腿闪光灯*)
	%QX0.10						:=	water_pump_ctl_sign					;	(*水泵控制指示*)

	%QX0.15						:=	triger_no_drawback_sign			;	(*支腿未全缩指示*)
	%QX0.14						:=	leveled_sign							;	(*下车调平指示*)
END_PROGRAM

(* POU I_O_CONFIGURATION/VEHICLE/io_config_10012, FBD *)
PROGRAM io_config_10012
VAR
	CH_NO1: INPUT_ANALOG;
	CH_NO2: INPUT_ANALOG;
	CH_NO3: INPUT_ANALOG;
	CH_NO4: INPUT_ANALOG;
	CH_NO5: FREQUENCY_E;
	CH_NO6: INPUT_ANALOG;



END_VAR
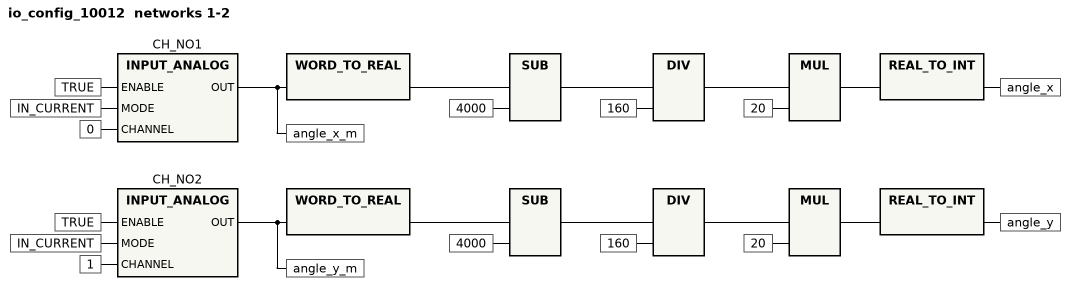
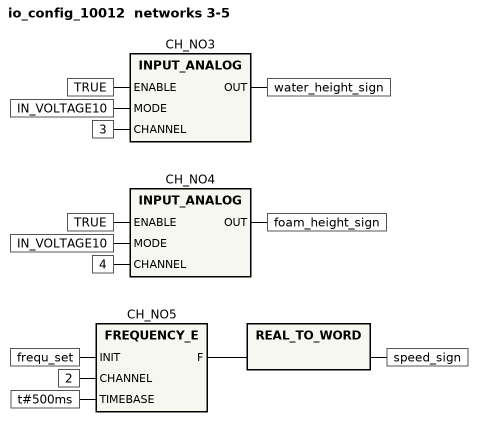
_FBD_ (* Function Block Diagram *)
NETWORK 1
	REAL_TO_INT(MUL(DIV(SUB(WORD_TO_REAL(<CH_NO1:INPUT_ANALOG(ENABLE: TRUE, MODE: IN_CURRENT, CHANNEL: 0) => angle_x_m>), 4000), 160), 20)) => angle_x
NETWORK 2
	REAL_TO_INT(MUL(DIV(SUB(WORD_TO_REAL(<CH_NO2:INPUT_ANALOG(ENABLE: TRUE, MODE: IN_CURRENT, CHANNEL: 1) => angle_y_m>), 4000), 160), 20)) => angle_y
NETWORK 3
	CH_NO3:INPUT_ANALOG(ENABLE: TRUE, MODE: IN_VOLTAGE10, CHANNEL: 3) => water_height_sign
NETWORK 4
	CH_NO4:INPUT_ANALOG(ENABLE: TRUE, MODE: IN_VOLTAGE10, CHANNEL: 4) => foam_height_sign
NETWORK 5
	REAL_TO_WORD(CH_NO5:FREQUENCY_E(INIT: frequ_set, CHANNEL: 2, TIMEBASE: t#500ms)) => speed_sign
_END_FBD_
(* the same logic as Structured Text *)
(* Network 1 *)
CH_NO1(ENABLE := TRUE, MODE := IN_CURRENT, CHANNEL := 0);
angle_x_m := CH_NO1.OUT;
angle_x := REAL_TO_INT(((WORD_TO_REAL(CH_NO1.OUT) - 4000) / 160) * 20);
(* Network 2 *)
CH_NO2(ENABLE := TRUE, MODE := IN_CURRENT, CHANNEL := 1);
angle_y_m := CH_NO2.OUT;
angle_y := REAL_TO_INT(((WORD_TO_REAL(CH_NO2.OUT) - 4000) / 160) * 20);
(* Network 3 *)
CH_NO3(ENABLE := TRUE, MODE := IN_VOLTAGE10, CHANNEL := 3);
water_height_sign := CH_NO3.OUT;
(* Network 4 *)
CH_NO4(ENABLE := TRUE, MODE := IN_VOLTAGE10, CHANNEL := 4);
foam_height_sign := CH_NO4.OUT;
(* Network 5 *)
CH_NO5(INIT := frequ_set, CHANNEL := 2, TIMEBASE := t#500ms);
speed_sign := REAL_TO_WORD(CH_NO5.F);
END_PROGRAM

(* POU I_O_CONFIGURATION/VEHICLE/io_config_address_10013, ST *)
PROGRAM io_config_address_10013
VAR
END_VAR
	front_left_Lv_ex_check1		:= %IX0.6			;	(*左前水平伸到位*)
	front_right_Lv_ex_check1		:= %IX0.7			;	(*右前水平伸到位*)
	back_left_Lv_ex_check1		:= %IX0.12			;	(*左后水平伸到位*)
	back_right_Lv_ex_check1	:= %IX0.13			;	(*右后水平伸到位*)
	front_left_urt_ex_check1		:= %IX0.14			;	(*左前垂直伸到位*)
	front_right_urt_ex_check1	:= %IX0.15			;	(*右前垂直伸到位*)
	back_left_urt_ex_check1		:= %IX1.4			;	(*左后垂直伸到位*)
	back_right_urt_ex_check1	:= %IX1.5			;	(*右后垂直伸到位*)

	front_left_Lv_drb_check		:= %IX32.1			;	(*左前水平收到位*)
	front_right_Lv_drb_check		:= %IX32.2			;	(*右前水平收到位*)
	back_left_Lv_drb_check		:= %IX32.3			;	(*左后水平收到位*)
	back_right_Lv_drb_check	:= %IX32.4			;	(*右后水平收到位*)
	front_left_urt_drb_check1		:= %IX32.5			;	(*左前垂直收到位*)
	front_right_urt_drb_check1	:= %IX32.6			;	(*右前垂直收到位*)
	back_left_urt_drb_check1	:= %IX32.7			;	(*左后垂直收到位*)
	back_right_urt_drb_check1	:= %IX32.12		;	(*右后垂直收到位*)

	engine_run					:= %IX2.2			;	(*发动机启动*)
	engine_stop					:= %IX2.3			;	(*发动机停止*)
	accelerate_sb					:= %IX2.0			;	(*加速*)
	decelerate_sb					:= %IX2.1			;	(*减速*)

(***操作***)
	tt_forcexx						:= %IX34.6			;	(*转台强制*)
	down_force					:= %IX34.7			;	(*下车强制*)
	auto_manu_choice			:= %IX34.1			;	(*自动/手动*)
	water_pump_run_sb			:= %IX1.7			;	(*消防泵开*)








	arm_to_station				:= %IX2.4			;	(*臂架到位检测*)
	water_pump_check			:= %IX33.4			;	(*水泵取力*)
	left_groud_check1			:= %IX34.4			;	(*车胎离地1*)
	left_groud_check2			:= %IX34.5			;	(*车胎离地2*)

	%QX32.2						:=	left_front_lv_ex_valve					;	(*左前水平伸*)
 	%QX32.0 						:=	left_back_lv_ex_valve					;	(*左后水平伸*)
 	%QX32.6						:=	right_front_lv_ex_valve				;	(*右前水平伸*)
	%QX32.4						:=	right_back_lv_ex_valve				;	(*右后水平伸*)
	%QX32.3						:=	left_front_lv_drb_valve				;	(*左前水平收*)
	%QX32.1						:=	left_back_lv_drb_valve				;	(*左后水平收*)
	%QX32.7						:=	right_front_lv_drb_valve				;	(*右前水平收*)
 	%QX32.5						:=	right_back_lv_drb_valve				;	(*右后水平收*)

(***底盘***)
	%QX0.8						:=	enginer_run_ctl						;	(*启动控制*)
	%QX0.9						:=	enginer_stop_ctl						;	(*熄火控制*)
 	%QX32.9						:=	enginer_acc_ctl						;	(*加速控制*)
	%QX32.10						:=	enginer_dec_ctl						;	(*减速控制*)

(***操作***)
	%QX0.10						:=	water_pump_ctl						;	(*水泵控制*)
	%QX32.14						:=	up_valve_ctl							;	(*上车阀*)
	%QX32.15						:=	down_valve_ctl						;	(*下车阀*)

(***指示***)
	%QX0.11						:=	over_level_sign						;	(*坡度超限*)
	%QX0.12						:=	triger_left_grd_sign					;	(*支腿离地*)
	%QX32.8						:=	alarmer_horn							;	(*警报器*)
	%QX32.13						:=	triger_flash							;	(*支腿闪光灯*)
	%QX0.10						:=	water_pump_ctl_sign					;	(*水泵控制指示*)

	%QX0.15						:=	triger_no_drawback_sign			;	(*支腿未全缩指示*)
	%QX0.14						:=	leveled_sign							;	(*下车调平指示*)
END_PROGRAM

(* POU I_O_CONFIGURATION/VEHICLE/io_config_10013, FBD *)
PROGRAM io_config_10013
VAR
	CH_NO1: INPUT_ANALOG;
	CH_NO2: INPUT_ANALOG;
	CH_NO3: INPUT_ANALOG;
	CH_NO4: INPUT_ANALOG;
	CH_NO5: FREQUENCY_E;
	CH_NO6: INPUT_ANALOG;



END_VAR
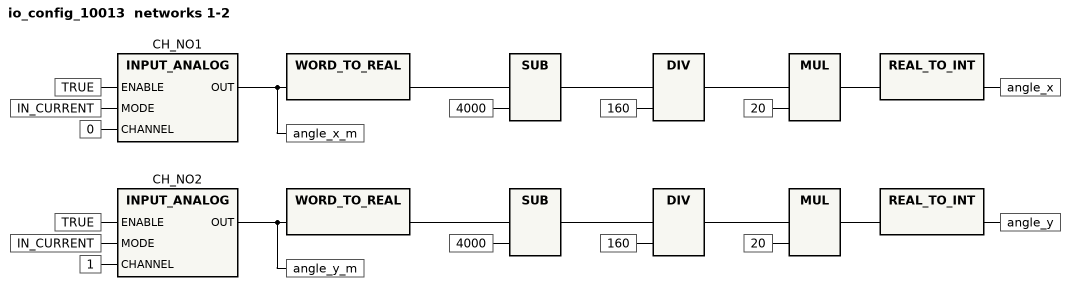
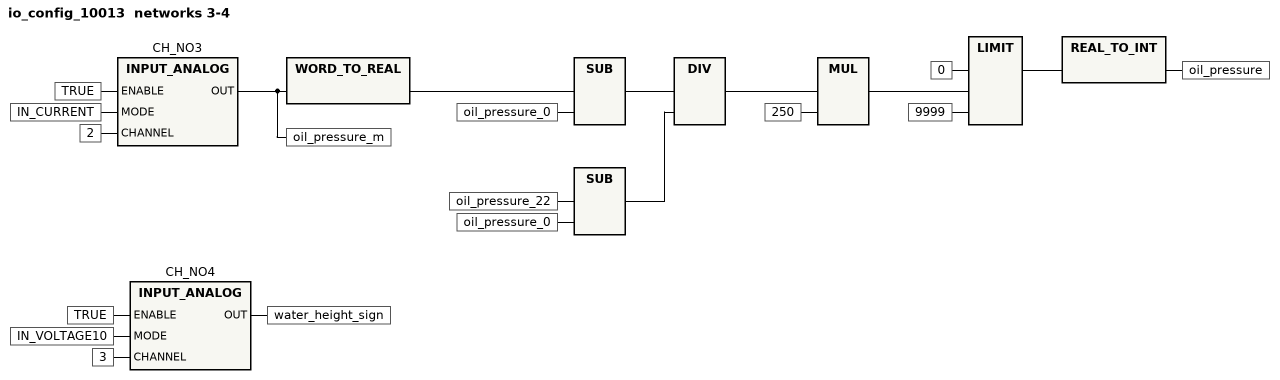
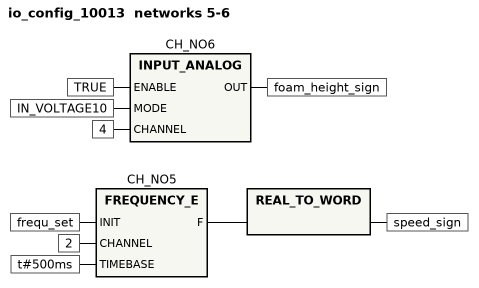
_FBD_ (* Function Block Diagram *)
NETWORK 1
	REAL_TO_INT(MUL(DIV(SUB(WORD_TO_REAL(<CH_NO1:INPUT_ANALOG(ENABLE: TRUE, MODE: IN_CURRENT, CHANNEL: 0) => angle_x_m>), 4000), 160), 20)) => angle_x
NETWORK 2
	REAL_TO_INT(MUL(DIV(SUB(WORD_TO_REAL(<CH_NO2:INPUT_ANALOG(ENABLE: TRUE, MODE: IN_CURRENT, CHANNEL: 1) => angle_y_m>), 4000), 160), 20)) => angle_y
NETWORK 3
	REAL_TO_INT(LIMIT(0, MUL(DIV(SUB(WORD_TO_REAL(<CH_NO3:INPUT_ANALOG(ENABLE: TRUE, MODE: IN_CURRENT, CHANNEL: 2) => oil_pressure_m>), oil_pressure_0), SUB(oil_pressure_22, oil_pressure_0)), 250), 9999)) => oil_pressure
NETWORK 4
	CH_NO4:INPUT_ANALOG(ENABLE: TRUE, MODE: IN_VOLTAGE10, CHANNEL: 3) => water_height_sign
NETWORK 5
	CH_NO6:INPUT_ANALOG(ENABLE: TRUE, MODE: IN_VOLTAGE10, CHANNEL: 4) => foam_height_sign
NETWORK 6
	REAL_TO_WORD(CH_NO5:FREQUENCY_E(INIT: frequ_set, CHANNEL: 2, TIMEBASE: t#500ms)) => speed_sign
_END_FBD_
(* the same logic as Structured Text *)
(* Network 1 *)
CH_NO1(ENABLE := TRUE, MODE := IN_CURRENT, CHANNEL := 0);
angle_x_m := CH_NO1.OUT;
angle_x := REAL_TO_INT(((WORD_TO_REAL(CH_NO1.OUT) - 4000) / 160) * 20);
(* Network 2 *)
CH_NO2(ENABLE := TRUE, MODE := IN_CURRENT, CHANNEL := 1);
angle_y_m := CH_NO2.OUT;
angle_y := REAL_TO_INT(((WORD_TO_REAL(CH_NO2.OUT) - 4000) / 160) * 20);
(* Network 3 *)
CH_NO3(ENABLE := TRUE, MODE := IN_CURRENT, CHANNEL := 2);
oil_pressure_m := CH_NO3.OUT;
oil_pressure := REAL_TO_INT(LIMIT(0, ((WORD_TO_REAL(CH_NO3.OUT) - oil_pressure_0) / (oil_pressure_22 - oil_pressure_0)) * 250, 9999));
(* Network 4 *)
CH_NO4(ENABLE := TRUE, MODE := IN_VOLTAGE10, CHANNEL := 3);
water_height_sign := CH_NO4.OUT;
(* Network 5 *)
CH_NO6(ENABLE := TRUE, MODE := IN_VOLTAGE10, CHANNEL := 4);
foam_height_sign := CH_NO6.OUT;
(* Network 6 *)
CH_NO5(INIT := frequ_set, CHANNEL := 2, TIMEBASE := t#500ms);
speed_sign := REAL_TO_WORD(CH_NO5.F);
END_PROGRAM

(* POU I_O_CONFIGURATION/VEHICLE/io_config_address_10014, ST *)
PROGRAM io_config_address_10014
VAR
END_VAR
	front_left_Lv_ex_check1		:= %IX0.6			;	(*左前水平伸到位*)
	front_right_Lv_ex_check1		:= %IX0.7			;	(*右前水平伸到位*)
	back_left_Lv_ex_check1		:= %IX0.12			;	(*左后水平伸到位*)
	back_right_Lv_ex_check1	:= %IX0.13			;	(*右后水平伸到位*)
	front_left_urt_ex_check1		:= %IX0.14			;	(*左前垂直伸到位*)
	front_right_urt_ex_check1	:= %IX0.15			;	(*右前垂直伸到位*)
	back_left_urt_ex_check1		:= %IX1.4			;	(*左后垂直伸到位*)
	back_right_urt_ex_check1	:= %IX1.5			;	(*右后垂直伸到位*)

	front_left_Lv_drb_check		:= %IX32.1			;	(*左前水平收到位*)
	front_right_Lv_drb_check		:= %IX32.2			;	(*右前水平收到位*)
	back_left_Lv_drb_check		:= %IX32.3			;	(*左后水平收到位*)
	back_right_Lv_drb_check	:= %IX32.4			;	(*右后水平收到位*)
	front_left_urt_drb_check1		:= %IX32.5			;	(*左前垂直收到位*)
	front_right_urt_drb_check1	:= %IX32.6			;	(*右前垂直收到位*)
	back_left_urt_drb_check1	:= %IX32.7			;	(*左后垂直收到位*)
	back_right_urt_drb_check1	:= %IX32.12		;	(*右后垂直收到位*)

	engine_run					:= %IX1.10			;	(*发动机启动*)
	engine_stop					:= %IX1.11			;	(*发动机停止*)
	accelerate_sb					:= %IX1.8			;	(*加速*)
	decelerate_sb					:= %IX1.9			;	(*减速*)

(***操作***)
	tt_forcexx						:= %IX33.14		;	(*转台强制*)
	down_force					:= %IX33.15		;	(*下车强制*)
	auto_manu_choice			:= %IX33.5			;	(*自动/手动*)
	water_pump_run_sb			:= %IX1.7			;	(*消防泵开*)








	arm_to_station				:= %IX1.12			;	(*臂架到位检测*)

	left_groud_check1			:= %IX33.12		;	(*车胎离地1*)
	left_groud_check2			:= %IX33.13		;	(*车胎离地2*)

	%QX32.2						:=	left_front_lv_ex_valve					;	(*左前水平伸*)
 	%QX32.0 						:=	left_back_lv_ex_valve					;	(*左后水平伸*)
 	%QX32.6						:=	right_front_lv_ex_valve				;	(*右前水平伸*)
	%QX32.4						:=	right_back_lv_ex_valve				;	(*右后水平伸*)
	%QX32.3						:=	left_front_lv_drb_valve				;	(*左前水平收*)
	%QX32.1						:=	left_back_lv_drb_valve				;	(*左后水平收*)
	%QX32.7						:=	right_front_lv_drb_valve				;	(*右前水平收*)
 	%QX32.5						:=	right_back_lv_drb_valve				;	(*右后水平收*)

(***底盘***)
	%QX1.0						:=	enginer_run_ctl						;	(*启动控制*)
	%QX1.1						:=	enginer_stop_ctl						;	(*熄火控制*)
 	%QX33.1						:=	enginer_acc_ctl						;	(*加速控制*)
	%QX33.2						:=	enginer_dec_ctl						;	(*减速控制*)

(***操作***)
	%QX1.2						:=	water_pump_ctl						;	(*水泵控制*)
	%QX33.6						:=	up_valve_ctl							;	(*上车阀*)
	%QX33.7						:=	down_valve_ctl						;	(*下车阀*)

(***指示***)
	%QX1.3						:=	over_level_sign						;	(*坡度超限*)
	%QX1.4						:=	triger_left_grd_sign					;	(*支腿离地*)
	%QX33.0						:=	alarmer_horn							;	(*警报器*)
	%QX33.5						:=	triger_flash							;	(*支腿闪光灯*)


	%QX1.6						:=	triger_no_drawback_sign			;	(*支腿未全缩指示*)
	%QX1.5						:=	leveled_sign							;	(*下车调平指示*)
END_PROGRAM

(* POU I_O_CONFIGURATION/VEHICLE/io_config_10014, FBD *)
PROGRAM io_config_10014
VAR
	CH_NO1: INPUT_ANALOG;
	CH_NO2: INPUT_ANALOG;
	CH_NO3: INPUT_ANALOG;
	CH_NO4: INPUT_ANALOG;
	CH_NO5: FREQUENCY_E;
	CH_NO6: INPUT_ANALOG;



END_VAR
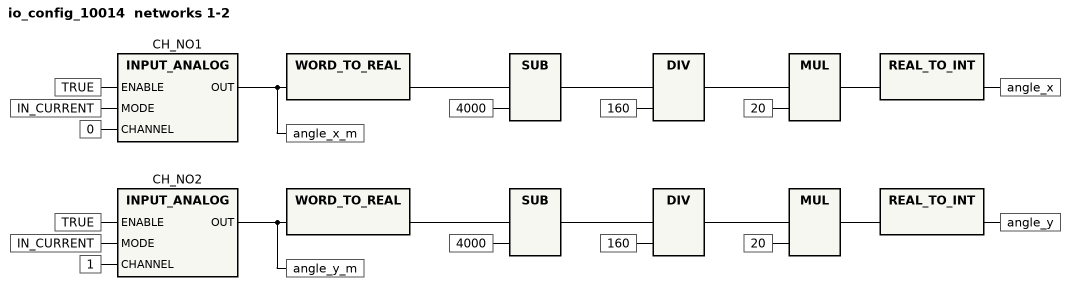
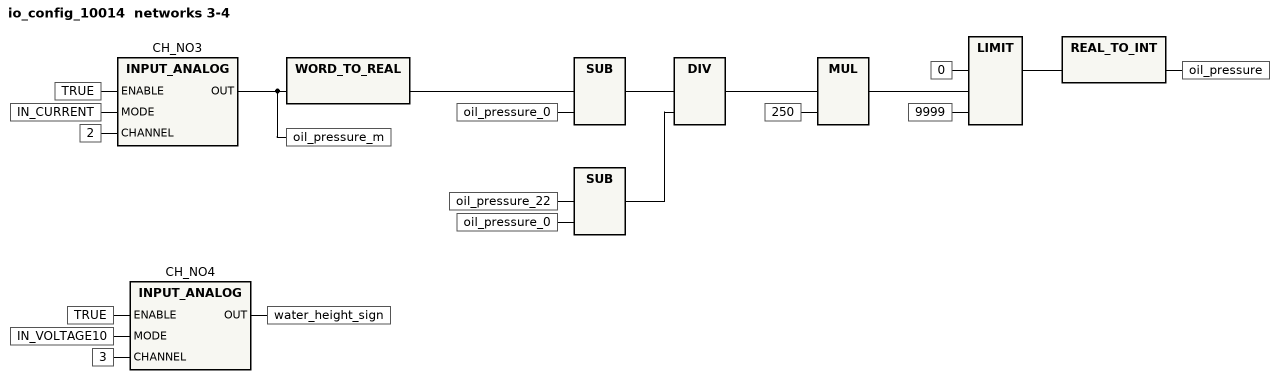
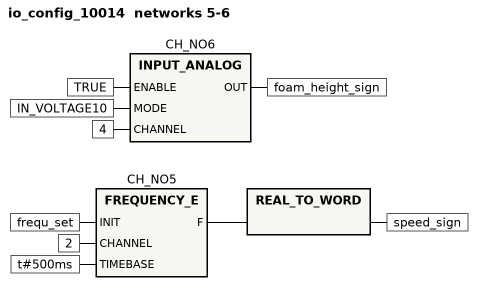
_FBD_ (* Function Block Diagram *)
NETWORK 1
	REAL_TO_INT(MUL(DIV(SUB(WORD_TO_REAL(<CH_NO1:INPUT_ANALOG(ENABLE: TRUE, MODE: IN_CURRENT, CHANNEL: 0) => angle_x_m>), 4000), 160), 20)) => angle_x
NETWORK 2
	REAL_TO_INT(MUL(DIV(SUB(WORD_TO_REAL(<CH_NO2:INPUT_ANALOG(ENABLE: TRUE, MODE: IN_CURRENT, CHANNEL: 1) => angle_y_m>), 4000), 160), 20)) => angle_y
NETWORK 3
	REAL_TO_INT(LIMIT(0, MUL(DIV(SUB(WORD_TO_REAL(<CH_NO3:INPUT_ANALOG(ENABLE: TRUE, MODE: IN_CURRENT, CHANNEL: 2) => oil_pressure_m>), oil_pressure_0), SUB(oil_pressure_22, oil_pressure_0)), 250), 9999)) => oil_pressure
NETWORK 4
	CH_NO4:INPUT_ANALOG(ENABLE: TRUE, MODE: IN_VOLTAGE10, CHANNEL: 3) => water_height_sign
NETWORK 5
	CH_NO6:INPUT_ANALOG(ENABLE: TRUE, MODE: IN_VOLTAGE10, CHANNEL: 4) => foam_height_sign
NETWORK 6
	REAL_TO_WORD(CH_NO5:FREQUENCY_E(INIT: frequ_set, CHANNEL: 2, TIMEBASE: t#500ms)) => speed_sign
_END_FBD_
(* the same logic as Structured Text *)
(* Network 1 *)
CH_NO1(ENABLE := TRUE, MODE := IN_CURRENT, CHANNEL := 0);
angle_x_m := CH_NO1.OUT;
angle_x := REAL_TO_INT(((WORD_TO_REAL(CH_NO1.OUT) - 4000) / 160) * 20);
(* Network 2 *)
CH_NO2(ENABLE := TRUE, MODE := IN_CURRENT, CHANNEL := 1);
angle_y_m := CH_NO2.OUT;
angle_y := REAL_TO_INT(((WORD_TO_REAL(CH_NO2.OUT) - 4000) / 160) * 20);
(* Network 3 *)
CH_NO3(ENABLE := TRUE, MODE := IN_CURRENT, CHANNEL := 2);
oil_pressure_m := CH_NO3.OUT;
oil_pressure := REAL_TO_INT(LIMIT(0, ((WORD_TO_REAL(CH_NO3.OUT) - oil_pressure_0) / (oil_pressure_22 - oil_pressure_0)) * 250, 9999));
(* Network 4 *)
CH_NO4(ENABLE := TRUE, MODE := IN_VOLTAGE10, CHANNEL := 3);
water_height_sign := CH_NO4.OUT;
(* Network 5 *)
CH_NO6(ENABLE := TRUE, MODE := IN_VOLTAGE10, CHANNEL := 4);
foam_height_sign := CH_NO6.OUT;
(* Network 6 *)
CH_NO5(INIT := frequ_set, CHANNEL := 2, TIMEBASE := t#500ms);
speed_sign := REAL_TO_WORD(CH_NO5.F);
END_PROGRAM

(* POU UNDER_DEALING/SPEED_ACT/VEHICLE/SPEED_ASSIGN, ST *)
(**************************限速*************************)
(*YT32*)				(*1300*)
(*YT32A*)				(*1400*)
(*YT32C*)				(*1700*)
(*YT32D*)				(*1700*)
(*YT32C旧版*)			(*1700*)
(*YT32D旧版*)			(*1700*)
(*YT32E*)				(*1400*)
(*YT32F*)				(*1400*)
(*YT32G*)				(*1700*)
(*YT32G旧版*)			(*1700*)
(*YT32H*)				(*1300*)
(*YT32J*)				(*1300*)
(*YT32K*)				(*1400*)
(*YT32L*)				(*1500*)
(*YT32M*)				(*1400*)
(*YT32N*)				(*1300*)


PROGRAM SPEED_ASSIGN
VAR


	ton1: TON;
	ton2: TON;
	ton3: TON;
	delay_set: BOOL;
	delay_set1: BOOL;
	delay_set2: BOOL;

	speed_r:R_TRIG;



	cruise_sign_set_t: TON;
END_VAR
CASE vehicle_styel OF
10011:
	vehicle_speed_10011();
10012:
	vehicle_speed_10012();
10013:
	vehicle_speed_10013();
10014:
	vehicle_speed_10014();
ELSE
	vehicle_speed_10013();
END_CASE


cruise_sign_set_t(in:=1,pt:=t#2s);
IF cruise_sign_set_t.Q THEN cruise_sign_set:=1;END_IF
IF leveled AND ((NOT up_down_switch AND tt_foot_switch) OR (up_down_switch AND stage_foot_switch)) THEN high_speed_set1:=1; ELSE   high_speed_set1:=0;END_IF
IF  NOT water_pump_ctl  AND cruise_sign_set  AND speed_sign>135 THEN
	IF (NOT withdraw_do AND NOT extend_do  AND NOT high_speed_set1 AND NOT extend_left_lv_triger_act AND NOT extend_right_lv_triger_act) OR (extend_do AND (extend_step=4 OR extend_step=5 OR extend_step=0)) THEN
		IF NOT delay_set2 THEN
			ton1(in:=1,pt:=t#700ms);enginer_acc_ctl:=0;	enginer_dec_ctl:=0;IF ton1.Q THEN delay_set2:=1;ton1(in:=0);END_IF
		ELSE
			low_speed_act();
		END_IF
	ELSE
		 delay_set2:=0;
	END_IF
	IF high_speed_set1 THEN
		IF NOT high_speed_set THEN
			ton2(in:=1,pt:=t#700ms);enginer_acc_ctl:=0;	enginer_dec_ctl:=0; IF ton2.Q THEN high_speed_set:=1;ton2(in:=0);END_IF
		ELSE
			up_speed_act();
		END_IF
	ELSE
		 high_speed_set:=0;
	END_IF
	IF (extend_do AND (extend_step=1 OR extend_step=2 OR extend_step=3 OR extend_step=6) ) OR withdraw_do OR extend_left_lv_triger_act OR extend_right_lv_triger_act THEN
		IF NOT delay_set1 THEN
			ton3(in:=1,pt:=t#700ms);enginer_acc_ctl:=0;	enginer_dec_ctl:=0;IF ton3.Q THEN delay_set1:=1;ton3(in:=0);END_IF
		ELSE
			down_speed_act();
		END_IF
	ELSE
		 delay_set1:=0;
	END_IF
END_IF
IF NOT cruise_sign_set THEN
	enginer_acc_ctl:=0;
	enginer_dec_ctl:=0;
END_IF
END_PROGRAM
ACTION vehicle_speed_10011:
(*
speed_r(clk:=speed_sel);
IF speed_r.Q THEN speed_l:=NOT speed_l; END_IF
IF speed_l THEN
	work_speed_l			:= 442;
	work_speed_h		:= 466;
	low_speed_l			:= 230;
	low_speed_h			:=280;
	high_speed_l			:=342;
	high_speed_h		:=392;
ELSE
	work_speed_l			:=270;
	work_speed_h		:=300;
	low_speed_l			:= 135;
	low_speed_h			:=178;
	high_speed_l			:=220;
	high_speed_h		:=250;
END_IF
*)
(*2.75倍 1300=472*)

	speed_m:=WORD_TO_REAL(speed_sign);
	speed_m:=speed_m*0.62;

	work_speed_l			:=442;
	work_speed_h		:=502;
	low_speed_l			:= 225;
	low_speed_h			:=285;
	high_speed_l			:=442;
	high_speed_h		:=502;
END_ACTION
ACTION vehicle_speed_10012:
(*
speed_r(clk:=speed_sel);
IF speed_r.Q THEN speed_l:=NOT speed_l; END_IF
IF speed_l THEN
	work_speed_l			:= 442;
	work_speed_h		:= 466;
	low_speed_l			:= 230;
	low_speed_h			:=280;
	high_speed_l			:=342;
	high_speed_h		:=392;
ELSE
	work_speed_l			:=270;
	work_speed_h		:=300;
	low_speed_l			:= 135;
	low_speed_h			:=178;
	high_speed_l			:=220;
	high_speed_h		:=250;
END_IF
*)
(*2.75倍 1300=472*)

	speed_m:=WORD_TO_REAL(speed_sign);
	speed_m:=speed_m*0.55;


	work_speed_l			:=520;
	work_speed_h		:=600;
	low_speed_l			:= 210;
	low_speed_h			:=270;
	high_speed_l			:=520;
	high_speed_h		:=600;
END_ACTION
ACTION vehicle_speed_10013:
(*
speed_r(clk:=speed_sel);
IF speed_r.Q THEN speed_l:=NOT speed_l; END_IF
IF speed_l THEN
	work_speed_l			:= 442;
	work_speed_h		:= 466;
	low_speed_l			:= 230;
	low_speed_h			:=280;
	high_speed_l			:=342;
	high_speed_h		:=392;
ELSE
	work_speed_l			:=270;
	work_speed_h		:=300;
	low_speed_l			:= 135;
	low_speed_h			:=178;
	high_speed_l			:=220;
	high_speed_h		:=250;
END_IF
*)
(*2.75倍 1300=472*)

	speed_m:=WORD_TO_REAL(speed_sign);
	speed_m:=speed_m*0.62;

	work_speed_l			:=442;
	work_speed_h		:=502;
	low_speed_l			:= 225;
	low_speed_h			:=285;
	high_speed_l			:=442;
	high_speed_h		:=502;
END_ACTION
ACTION vehicle_speed_10014:
(*
speed_r(clk:=speed_sel);
IF speed_r.Q THEN speed_l:=NOT speed_l; END_IF
IF speed_l THEN
	work_speed_l			:= 442;
	work_speed_h		:= 466;
	low_speed_l			:= 230;
	low_speed_h			:=280;
	high_speed_l			:=342;
	high_speed_h		:=392;
ELSE
	work_speed_l			:=270;
	work_speed_h		:=300;
	low_speed_l			:= 135;
	low_speed_h			:=178;
	high_speed_l			:=220;
	high_speed_h		:=250;
END_IF
*)
(*2.75倍 1300=472*)

	speed_m:=WORD_TO_REAL(speed_sign);
	speed_m:=speed_m*0.62;

	work_speed_l			:=442;
	work_speed_h		:=502;
	low_speed_l			:= 225;
	low_speed_h			:=285;
	high_speed_l			:=442;
	high_speed_h		:=502;
END_ACTION

(* POU UNDER_DEALING/SPEED_ACT/low_speed_act, ST *)
PROGRAM low_speed_act
VAR
END_VAR
IF speed_sign<=low_speed_l  THEN
	enginer_acc_ctl:=1;
	enginer_dec_ctl:=0;
END_IF
IF speed_sign>=low_speed_h  THEN
	enginer_acc_ctl:=0;
	enginer_dec_ctl:=1;
END_IF
IF speed_sign>=low_speed_l AND speed_sign<=low_speed_h THEN
	enginer_acc_ctl:=0;
	enginer_dec_ctl:=0;
END_IF
END_PROGRAM

(* POU UNDER_DEALING/SPEED_ACT/up_speed_act, ST *)
PROGRAM up_speed_act
VAR
END_VAR
IF speed_sign<=work_speed_l  THEN
	enginer_acc_ctl:=1;
	enginer_dec_ctl:=0;
END_IF
IF speed_sign>=work_speed_h  THEN
	enginer_acc_ctl:=0;
	enginer_dec_ctl:=1;
END_IF
IF speed_sign>=work_speed_l AND speed_sign<=work_speed_h THEN
	enginer_acc_ctl:=0;
	enginer_dec_ctl:=0;
END_IF
END_PROGRAM

(* POU UNDER_DEALING/SPEED_ACT/down_speed_act, ST *)
PROGRAM down_speed_act
VAR
END_VAR
IF speed_sign<=high_speed_l  THEN
	enginer_acc_ctl:=1;
	enginer_dec_ctl:=0;
END_IF
IF speed_sign>=high_speed_h  THEN
	enginer_acc_ctl:=0;
	enginer_dec_ctl:=1;
END_IF
IF speed_sign>=high_speed_l AND speed_sign<=high_speed_h THEN
	enginer_acc_ctl:=0;
	enginer_dec_ctl:=0;
END_IF
END_PROGRAM

(* POU TRIGER_LEVEL/VEHICLE/LEVEL, ST *)
PROGRAM LEVEL

VAR_INPUT
	init1: INT;
END_VAR

VAR_OUTPUT
	a: INT;
END_VAR

VAR

END_VAR
left_front_lv_ex_valve					:=0;
right_front_lv_ex_valve				:=0;
left_back_lv_ex_valve					:=0;
right_back_lv_ex_valve				:=0;
left_front_lv_drb_valve				:=0;
left_back_lv_drb_valve				:=0;
right_front_lv_drb_valve				:=0;
right_back_lv_drb_valve				:=0;
left_front_desired						:=0;
right_front_desired					:=0;
left_back_desired						:=0;
right_back_desired					:=0;
left_front_drawback_desired			:=0;
right_front_drawback_desired		:=0;
left_back_drawback_desired			:=0;
right_back_drawback_desired		:=0;

leg_check_deal();
leg_check_auto();


levelling();
LEVEL_PROMPT();

CASE vehicle_styel OF
10011:
	levelling2_remote2();
10012,10013,10014:
	levelling2_remote();
ELSE
	levelling2_remote2();
END_CASE

triger_pwm();
END_PROGRAM

(* POU TRIGER_LEVEL/leg_check_deal, ST *)
PROGRAM leg_check_deal
VAR

	back_left_ton_L: TON;
	back_right_ton_L:TON;
	front_left_ton_L:TON;
	front_right_ton_L:TON;

	back_left_ton: TON;
	back_right_ton:TON;
	front_left_ton:TON;
	front_right_ton:TON;

END_VAR
(*************水平开关延时****************************************************************)
front_left_ton_L(in:=front_left_Lv_ex_check1,pt:=t#2000ms);
front_left_Lv_ex_check:=front_left_ton_L.Q;

front_right_ton_L(in:=front_right_Lv_ex_check1,pt:=t#2000ms);
front_right_Lv_ex_check:=front_right_ton_L.Q;

back_left_ton_L(in:=back_left_Lv_ex_check1,pt:=t#2000ms);
back_left_Lv_ex_check:=back_left_ton_L.Q;

back_right_ton_L(in:=back_right_Lv_ex_check1,pt:=t#2000ms);
back_right_Lv_ex_check:=back_right_ton_L.Q;

(***************垂直开关延时**************************************************************)
front_left_ton(in:= front_left_urt_ex_check1,pt:=t#1000ms);
front_left_urt_ex_check:=front_left_ton.Q;

front_right_ton(in:= front_right_urt_ex_check1,pt:=t#1000ms);
front_right_urt_ex_check:=front_right_ton.Q;

back_left_ton(in:= back_left_urt_ex_check1,pt:=t#1000ms);
back_left_urt_ex_check:=back_left_ton.Q;

back_right_ton(in:= back_right_urt_ex_check1,pt:=t#1000ms);
back_right_urt_ex_check:=back_right_ton.Q;


front_left_urt_drb_check			:=NOT front_left_urt_drb_check1;
front_right_urt_drb_check		:=NOT front_right_urt_drb_check1;
back_left_urt_drb_check			:=NOT back_left_urt_drb_check1;
back_right_urt_drb_check		:=NOT back_right_urt_drb_check1;
END_PROGRAM

(* POU TRIGER_LEVEL/leg_check_auto, ST *)
PROGRAM leg_check_auto
VAR

	v_touch_speed					:WORD := 500;

	i,j									:INT;
	leg_step							:INT;
	leg_step_t1						:TON;

	compare							:ARRAY [1..4,1..4]OF WORD;
	compare_w1						:WORD;
	compare_w2						:WORD;

	leg_test_R						:R_TRIG;
	front_left_urt_ex_check1_R		:R_TRIG;
	front_right_urt_ex_check1_R		:R_TRIG;
	back_left_urt_ex_check1_R		:R_TRIG;
	back_right_urt_ex_check1_R		:R_TRIG;

	front_left_urt_ex_m				:BOOL;
	front_right_urt_ex_m				:BOOL;
	back_left_urt_ex_m				:BOOL;
	back_right_urt_ex_m				:BOOL;

	time_read1						:TIMER_READ;

	front_left_urt_time				:TIME;
	front_left_urt_time1			:TIME;
	front_left_urt_time2			:TIME;
	front_right_urt_time			:TIME;
	front_right_urt_time1			:TIME;
	front_right_urt_time2			:TIME;
	back_left_urt_time			:TIME;
	back_left_urt_time1			:TIME;
	back_left_urt_time2			:TIME;
	back_right_urt_time			:TIME;
	back_right_urt_time1			:TIME;
	back_right_urt_time2			:TIME;



	a: BOOL;
	b: BOOL;
	c: BOOL;

	a_r:R_TRIG;
	b_r:R_TRIG;
	c_r:R_TRIG;

END_VAR
(*************************************************************************

前后支腿间距											6500
支腿离地高度（不考虑板簧下降）					504		车头朝下（6°    946   257）	（5°    871   298）		（4°    797   339）		（3°    724   380）	（2°    650   421）（1°    577   463）
																	车头朝上（6°    1373   684）	（5°    1227   654）	（4°    1082   624）	（3°    937   594）	（2°    792   564）（1°    648   534）
支腿间隙												50


*************************************************************************)





leg_test_R(CLK:=leg_test);

IF leg_test_R.Q THEN
		leg_test_m:=1;
		leg_step:=1;
		front_left_urt_time				:=t#0s;
		front_left_urt_time1			:=t#0s;
		front_left_urt_time2			:=t#0s;
		front_right_urt_time			:=t#0s;
		front_right_urt_time1			:=t#0s;
		front_right_urt_time2			:=t#0s;
		back_left_urt_time			:=t#0s;
		back_left_urt_time1			:=t#0s;
		back_left_urt_time2			:=t#0s;
		back_right_urt_time			:=t#0s;
		back_right_urt_time1			:=t#0s;
		back_right_urt_time2			:=t#0s;
END_IF

IF NOT arm_to_station THEN
		leg_test_m:=0;
		leg_step:=0;
END_IF


IF leg_test_m AND arm_to_station THEN
	IF(leg_step=1) THEN
		IF NOT front_left_urt_drb_check 		THEN left_front_drawback_desired:=500; 		ELSE	left_front_drawback_desired:=0;		END_IF
		IF NOT front_right_urt_drb_check 	THEN right_front_drawback_desired:=500;		ELSE	right_front_drawback_desired:=0; 	END_IF
		IF NOT back_left_urt_drb_check 		THEN left_back_drawback_desired:=500; 		ELSE	left_back_drawback_desired:=0;		END_IF
		IF NOT back_right_urt_drb_check	THEN right_back_drawback_desired:=500; 		ELSE	right_back_drawback_desired:=0;	END_IF
		leg_step_t1(in:= (front_left_urt_drb_check AND front_right_urt_drb_check AND back_left_urt_drb_check AND back_right_urt_drb_check),pt:=t#1s);
		IF leg_step_t1.Q THEN 	leg_step:=2; 	leg_step_t1(in:=0);	END_IF
	END_IF

	IF(leg_step=2) THEN
		IF NOT(front_left_Lv_ex_check) 		THEN		left_front_lv_ex_valve:=1;		ELSE		left_front_lv_ex_valve:=0;		END_IF
		IF NOT(front_right_Lv_ex_check) 	THEN		right_front_lv_ex_valve:=1;	ELSE		right_front_lv_ex_valve:=0;	END_IF
		IF NOT(back_left_Lv_ex_check) 		THEN		left_back_lv_ex_valve:=1;		ELSE		left_back_lv_ex_valve:=0;		END_IF
		IF NOT(back_right_Lv_ex_check) 	THEN		right_back_lv_ex_valve:=1;	ELSE		right_back_lv_ex_valve:=0;	END_IF

		IF front_left_Lv_ex_check AND front_right_Lv_ex_check AND back_left_Lv_ex_check AND back_right_Lv_ex_check THEN
			front_left_urt_time1			:=time_read1.T;
			front_right_urt_time1			:=time_read1.T;
			back_left_urt_time1			:=time_read1.T;
			back_right_urt_time1			:=time_read1.T;
			IF NOT front_left_urt_ex_check1 		AND  front_left_urt_ex_m 		THEN left_front_desired		:=v_touch_speed; 	ELSE left_front_desired:=0; 		END_IF
			IF NOT front_right_urt_ex_check1  	AND  front_right_urt_ex_m 	THEN right_front_desired	:=v_touch_speed; 	ELSE right_front_desired:=0; 	END_IF
			IF NOT back_left_urt_ex_check1 		AND  back_left_urt_ex_m 	THEN left_back_desired		:=v_touch_speed; 	ELSE left_back_desired:=0; 		END_IF
			IF NOT back_right_urt_ex_check1 	AND  back_right_urt_ex_m 	THEN right_back_desired	:=v_touch_speed; 	ELSE right_back_desired:=0; 	END_IF

			front_left_urt_ex_check1_R(CLK:=front_left_urt_ex_check1);
			front_right_urt_ex_check1_R(CLK:=front_right_urt_ex_check1);
			back_left_urt_ex_check1_R(CLK:=back_left_urt_ex_check1);
			back_right_urt_ex_check1_R(CLK:=back_right_urt_ex_check1);
	
			IF front_left_urt_ex_check1 		THEN 		left_front_desired:=0; 			front_left_urt_ex_m:=0;		END_IF
			IF front_right_urt_ex_check1 		THEN 		right_front_desired:=0; 		front_right_urt_ex_m:=0;		END_IF
			IF back_left_urt_ex_check1 		THEN 		right_front_desired:=0; 		back_left_urt_ex_m:=0;		END_IF
			IF back_right_urt_ex_check1 		THEN 		right_front_desired:=0; 		back_right_urt_ex_m:=0;		END_IF

			IF front_left_urt_ex_check1_R.Q		 THEN 		front_left_urt_time2	:=time_read1.T;		front_left_urt_time		:=front_left_urt_time1-front_left_urt_time2;		front_left_urt_time_W		:=TIME_TO_WORD(front_left_urt_time);		END_IF
			IF front_right_urt_ex_check1_R.Q 	THEN 		front_right_urt_time2	:=time_read1.T;		front_right_urt_time	:=front_right_urt_time1-front_right_urt_time2;	front_right_urt_time_W	:=TIME_TO_WORD(front_right_urt_time);	END_IF
			IF back_left_urt_ex_check1_R.Q 		THEN 		back_left_urt_time2	:=time_read1.T;		back_left_urt_time	:=back_left_urt_time1-back_left_urt_time2;		back_left_urt_time_W		:=TIME_TO_WORD(back_left_urt_time);		END_IF
			IF back_right_urt_ex_check1_R.Q 	THEN 		back_right_urt_time2	:=time_read1.T;		back_right_urt_time	:=back_right_urt_time1-back_right_urt_time2;	back_right_urt_time_W	:=TIME_TO_WORD(back_right_urt_time);	END_IF

			IF NOT (front_left_urt_time_W=0) AND NOT (front_right_urt_time_W=0) AND NOT (back_left_urt_time_W=0) AND NOT (back_right_urt_time_W=0)  THEN leg_step:=3; END_IF
		END_IF
	END_IF

	IF(leg_step=3) THEN
		compare[1,1]:=front_left_urt_time_W;
		compare[2,1]:=front_right_urt_time_W;
		compare[3,1]:=back_left_urt_time_W;
		compare[4,1]:=back_right_urt_time_W;
		compare[1,2]:=1;
		compare[2,2]:=2;
		compare[3,2]:=3;
		compare[4,2]:=4;

		FOR i:=1 TO 3 BY 1 DO
			FOR j:=1 TO 4-i BY 1 DO
				IF compare[j,1]>compare[j+1,1] THEN 	compare_w1:=compare[j,1]; 		compare[j,1]:=compare[j+1,1]; 	compare[j+1,1]:=compare_w1;
															compare_w2:=compare[j,2]; 		compare[j,2]:=compare[j+1,2]; 	compare[j+1,2]:=compare_w2;			END_IF
			END_FOR
		END_FOR

		IF ABS(compare[4,1]-compare[1,1])>2000 THEN
			IF  compare[4,2]=1 THEN fl_fac_nr:=fl_fac_nr-1; END_IF
			IF  compare[4,2]=2 THEN fr_fac_nr:=fr_fac_nr-1; END_IF
			IF  compare[4,2]=3 THEN rl_fac_nr:=rl_fac_nr-1; END_IF
			IF  compare[4,2]=4 THEN rr_fac_nr:=rr_fac_nr-1; END_IF
			front_left_urt_time				:=t#0s;
			front_left_urt_time1			:=t#0s;
			front_left_urt_time2			:=t#0s;
			front_right_urt_time			:=t#0s;
			front_right_urt_time1			:=t#0s;
			front_right_urt_time2			:=t#0s;
			back_left_urt_time			:=t#0s;
			back_left_urt_time1			:=t#0s;
			back_left_urt_time2			:=t#0s;
			back_right_urt_time			:=t#0s;
			back_right_urt_time1			:=t#0s;
			back_right_urt_time2			:=t#0s;
			front_left_urt_time_W			:=0;
			front_right_urt_time_W		:=0;
			back_left_urt_time_W			:=0;
			back_right_urt_time_W		:=0;
			leg_step:=1;
		ELSE
			leg_step:=0;
			leg_test_m:=0;
		END_IF
	END_IF

END_IF
END_PROGRAM

(* POU TRIGER_LEVEL/levelling, ST *)
PROGRAM levelling
VAR
	ton0				: TON;
	extend_act			: R_TRIG;
	ton1				: TON;
	ton1_2				: TON;
	angle_dir			: BYTE;
	tem2				: DINT;
	h_out_time		: INT := 30;
	left_ok				: BOOL;
	right_ok			: BOOL;
	v_touch_time		: INT := 48;
	fl_to_groud		: BOOL;
	fr_to_groud		: BOOL;
	bl_to_groud		: BOOL;
	br_to_groud		: BOOL;
	v_touch_speed	: WORD := 500;
	angle_x_real		: REAL;
	angle_x_offset_real: REAL;
	set_x				: WORD;
	angle_y_real		: REAL;
	angle_y_offset_real: REAL;
	set_y: WORD;
	angle_ok: INT := 50;
	PID_level: PID;
	set_x_real: REAL;
	PID_level_y: PID;
	set_y_real: REAL;
	x_limit: BOOL;
	y_limit: BOOL;
	v_rise_time: INT := 20;
	step_4_limit: WORD := 200;
	v_rise_speed: WORD := 100;
	prop_m_1: REAL := 1;
	prop_m: REAL := 1;
	ton_step4: TON;
	angle_ok_sign: INT;
	level_time: INT := 15;
	tontp: TON;
	v_in_speed: WORD := 500;
	drawback_act: R_TRIG;
	v_in_time: INT := 50;
	x_over: BOOL;
	y_over: BOOL;
	PD1: PD;
	PD2: PD;
	PD3: PD;
	PD4: PD;
	leave_ground_sign: BOOL;

	three_step:BOOL;
	side_l:BOOL;
	side_r:BOOL;
	side_m:BOOL;
	tona1:TON;
	tona2:TON;
	tona3:TON;
	tona4:TON;
       tona_m1:BOOL;
       tona_m2:BOOL;
       tona_m3:BOOL;
       tona_m4:BOOL;

	x1		: INT:=0;
	x2		: INT:=0;
	x3		: INT:=0;
	xm1: INT;
	xm2: INT;
	xm3: INT;
	xm4: INT;
	angle_x_a:ARRAY[0..14] OF INT;
	angle_y_a:ARRAY[0..14] OF INT;
	x_value	: INT;
	y_value	: INT;

	angle_x2: INT:=1000;
	angle_y2: INT :=1000;


	angle_y_r1: INT;
	angle_y_r2: INT;

	withdraw_fl:INT;
	withdraw_fr:INT;
	withdraw_bl:INT;
	withdraw_br:INT;

	angle_withdraw_x1: INT;
	angle_withdraw_y1: INT;
	angle_withdraw_x2: INT;
	angle_withdraw_y2: INT;
	withdraw_m1:BOOL;
	withdraw_m2:BOOL;
	withdraw_m3:BOOL;
	withdraw_m4:BOOL;
	withdraw_mx:INT;
	withdraw_my:INT;
	withdraw_t1:TON;
	withdraw_m5:BOOL;
	w_value:INT:=2;

	step2_m1:BOOL;
	step2_m2:BOOL;
	step2_m3:BOOL;
	step2_m4:BOOL;
	step2_m5:BOOL;
	step2_m6:BOOL;
	step4_m1:INT;
	step4_m2:INT;
	step4_m3:INT;
	step4_m4:INT;
	ton_withdraw:TON;

	level_second: BOOL;
	ton4_second:TON;
	ton6_yanshi:TON;

	extend_left_lv_triger_r: R_TRIG;
	extend_right_lv_triger_r: R_TRIG;

	ton_second:TON;
	allow_second: BOOL;


	angle_xx: INT;


	leg_time_int_m		:INT;
	leg_time_charcurve	:CHARCURVE;
	leg_time				:TIME:=t#9s;


END_VAR
(*************************************************清零***********************************************)
left_front_desired					:=0;
right_front_desired				:=0;
left_back_desired					:=0;
right_back_desired				:=0;
right_front_drawback_desired	:=0;
left_back_drawback_desired		:=0;
right_back_drawback_desired	:=0;
left_front_drawback_desired		:=0;
left_front_lv_ex_valve				:=0;
left_back_lv_ex_valve				:=0;
right_front_lv_ex_valve			:=0;
right_back_lv_ex_valve			:=0;
left_front_lv_drb_valve			:=0;
left_back_lv_drb_valve			:=0;
right_front_lv_drb_valve			:=0;
right_back_lv_drb_valve			:=0;

(**********sl************增加***平均值滤波*********15组值取5组*******start*)
	angle_x_a[x1]:=angle_x;
	angle_y_a[x1]:=angle_y;
	x1:=x1+1;
IF(x1>=14) THEN
	FOR x2:=0 TO 13 BY 1 DO
		x3:=0;
		FOR x3:=0 TO 13 BY 1 DO
			IF(angle_x_a[x3]<angle_x_a[x3+1]) THEN  xm1:=angle_x_a[x3+1];  angle_x_a[x3+1]:=angle_x_a[x3]; angle_x_a[x3]:=xm1; END_IF
			IF(angle_y_a[x3]<angle_y_a[x3+1]) THEN  xm2:=angle_y_a[x3+1];  angle_y_a[x3+1]:=angle_y_a[x3]; angle_y_a[x3]:=xm2; END_IF
		END_FOR
	END_FOR
	IF(x2>=13) THEN
		xm3:=angle_x_a[5]+angle_x_a[6]+angle_x_a[7]+angle_x_a[8]+angle_x_a[9];
		xm4:=angle_y_a[5]+angle_y_a[6]+angle_y_a[7]+angle_y_a[8]+angle_y_a[9];
		angle_x2:=xm3/5;
		angle_y2:=xm4/5;
		x1:=0;
	END_IF
END_IF
angle_x:=angle_x2;
angle_y:=angle_y2;

IF NOT (angle_y_r1=angle_y)THEN
	angle_y_r2:=angle_y_r1;
	angle_y_r1:=angle_y;
END_IF
(***********sl***********增加***平均值滤波*********15组值取5组*********end*)

(*
(*————————————————————————————自动支腿第一步————————————————————————————————————————*)
(*第一步：伸水平支腿*)
	IF extend_step=1 THEN
(*在伸水平支腿时关收水平支腿阀*)
		left_front_lv_drb_valve	:=0;
		left_back_lv_drb_valve	:=0;
		right_front_lv_drb_valve	:=0;
		right_back_lv_drb_valve 	:=0;
		tem2:=INT_TO_DINT(h_out_time)*1000;
		ton1(in:=1,pt:=DINT_TO_TIME(tem2));
		ton1;
(*左边的支腿水平处理*)
		IF (NOT right_side_choice AND  NOT left_side_choice)OR left_side_choice THEN
			IF NOT(front_left_Lv_ex_check) THEN
				left_front_lv_ex_valve:=1;
			ELSE
				left_front_lv_ex_valve:=0;
			END_IF
			IF NOT(back_left_Lv_ex_check) THEN
				left_back_lv_ex_valve:=1;
			ELSE
				left_back_lv_ex_valve:=0;
			END_IF
		END_IF
(*右边的支腿水平处理*)
		IF (NOT right_side_choice AND  NOT left_side_choice)OR right_side_choice THEN
			IF NOT(front_right_Lv_ex_check) THEN
				right_front_lv_ex_valve:=1;
			ELSE
				right_front_lv_ex_valve:=0;
			END_IF
			IF NOT(back_right_Lv_ex_check) THEN
				right_back_lv_ex_valve:=1;
			ELSE
				right_back_lv_ex_valve:=0;
			END_IF
		END_IF
	(*如果支腿伸到位或者右单边则左伸OK*)
		IF ((NOT right_side_choice)AND front_left_Lv_ex_check AND back_left_Lv_ex_check) OR right_side_choice THEN
			left_ok:=1;
		END_IF

	(*如果支腿伸到位或者左单边则右伸OK*)
		IF ((NOT left_side_choice)AND front_right_Lv_ex_check AND back_right_Lv_ex_check) OR left_side_choice THEN
			right_ok:=1;
		END_IF

(*支腿水平展开完毕后关闭水平阀*)
		IF (left_ok AND right_ok) OR ton1.q OR(front_left_Lv_ex_check AND back_left_Lv_ex_check AND front_right_Lv_ex_check AND back_right_Lv_ex_check) THEN
			ton1(in:=0);
			extend_step:=2;
			left_ok:=0;
			right_ok:=0;
			tona_m1:=1;
			tona_m2:=1;
			tona_m3:=1;
			tona_m4:=1;
		END_IF
(*四种倾角太大的情况*)
	END_IF
*)



(*伸水平支腿*)
extend_left_lv_triger_r(CLK:= level_extend_triger_left  AND auto_manu_choice AND arm_to_station AND( NOT leveled OR withdraw_do ));
extend_right_lv_triger_r(CLK:= level_extend_triger_right AND auto_manu_choice AND arm_to_station AND( NOT leveled OR withdraw_do ));
IF extend_left_lv_triger_r.Q 	THEN  extend_left_lv_triger_act:=NOT extend_left_lv_triger_act; 		END_IF
IF extend_right_lv_triger_r.Q 	THEN  extend_right_lv_triger_act:=NOT extend_right_lv_triger_act; 	END_IF
(*左*)
IF extend_left_lv_triger_act THEN
	withdraw_do:=0;
	extend_do:=0;
	left_front_lv_drb_valve	:=0;
	left_back_lv_drb_valve	:=0;
	right_front_lv_drb_valve	:=0;
	right_back_lv_drb_valve 	:=0;
	tem2:=INT_TO_DINT(h_out_time)*1000;
	ton1(in:=1,pt:=DINT_TO_TIME(tem2));
	ton1;
	IF NOT(front_left_Lv_ex_check) THEN
		left_front_lv_ex_valve:=1;
	ELSE
		left_front_lv_ex_valve:=0;
	END_IF
	IF NOT(back_left_Lv_ex_check) THEN
		left_back_lv_ex_valve:=1;
	ELSE
		left_back_lv_ex_valve:=0;
	END_IF
	IF (front_left_Lv_ex_check AND back_left_Lv_ex_check)OR ton1.q THEN  extend_left_lv_triger_act:=0; ton1(in:=0);END_IF
END_IF
(*右*)

IF extend_right_lv_triger_act THEN
	withdraw_do:=0;
	extend_do:=0;
	left_front_lv_drb_valve	:=0;
	left_back_lv_drb_valve	:=0;
	right_front_lv_drb_valve	:=0;
	right_back_lv_drb_valve 	:=0;
	tem2:=INT_TO_DINT(h_out_time)*1000;
	ton1_2(in:=1,pt:=DINT_TO_TIME(tem2));
	ton1;
	IF NOT(front_right_Lv_ex_check) THEN
		right_front_lv_ex_valve:=1;
	ELSE
		right_front_lv_ex_valve:=0;
	END_IF
	IF NOT(back_right_Lv_ex_check) THEN
		right_back_lv_ex_valve:=1;
	ELSE
		right_back_lv_ex_valve:=0;
	END_IF
	IF (front_right_Lv_ex_check AND back_right_Lv_ex_check )OR ton1_2.q THEN  extend_right_lv_triger_act:=0; ton1_2(in:=0);END_IF
END_IF


(*----------------------------------------------启动自动支腿--------------------------------------------------------*)
auto_extend_triger:=auto_extend_triger_left OR auto_extend_triger_right;
IF NOT leveled THEN level_second:=FALSE;END_IF
(*伸支腿操作*)
extend_act(CLK:= auto_extend_triger);
IF (extend_act.q) AND auto_manu_choice AND arm_to_station AND NOT extend_left_lv_triger_act AND NOT extend_right_lv_triger_act AND( (front_right_Lv_ex_check AND back_right_Lv_ex_check)OR(front_left_Lv_ex_check AND back_left_Lv_ex_check))THEN
	extend_do:=NOT extend_do;
	withdraw_do:=0;
	extend_left_lv_triger_act:=0;
	extend_right_lv_triger_act:=0;
	ton1(in:=0);ton6_yanshi(in:=0);ton4_second(in:=0);
	IF leveled THEN
		extend_step:=4;level_second:=TRUE;
	ELSE
	extend_step:=2;level_second:=FALSE;
	END_IF
(***********************sl**增加*****************************************start*)
	IF(extend_do AND NOT leveled)THEN
		IF(angle_y-angle_y_offset>=0)THEN head_b3:=1; head_f3:=0;  END_IF
		IF(angle_y-angle_y_offset<0)THEN head_f3:=1; head_b3:=0; END_IF
		IF(angle_y-angle_y_offset>50)THEN head_b:=1; head_f:=0;  END_IF
		IF(angle_y-angle_y_offset<-50)THEN head_f:=1; head_b:=0; END_IF
		IF(angle_y-angle_y_offset>150)THEN head_b2:=1; head_f2:=0;END_IF
		IF(angle_y-angle_y_offset<-150)THEN head_f2:=1; head_b2:=0;END_IF
		IF(angle_x-angle_x_offset>250)THEN side_r:=1; side_l:=0;END_IF
		IF(angle_x-angle_x_offset<-250)THEN side_l:=1; side_r:=0;END_IF
	END_IF

	IF head_b2 OR head_f2 THEN angle_ok:=75; ELSE angle_ok:=50; END_IF
(***********************sl**增加*******************************************end*)


(***********************sl**增加*****************************************start*)
IF angle_y-angle_y_offset>=0 	THEN	leg_time_charcurve(in:=(angle_y-angle_y_offset),n:=4,P:=ll_f,out=>leg_time_int_m);			END_IF
IF angle_y-angle_y_offset<0 		THEN	leg_time_charcurve(in:=-(angle_y-angle_y_offset),n:=4,P:=ll_b,out=>leg_time_int_m);		END_IF
(*
leg_time							:=REAL_TO_TIME(leg_time_int_m*(WORD_TO_REAL(front_left_urt_time_W))/504);
*)
(***********************sl**增加*******************************************end*)

END_IF

IF leveled THEN
	head_b3:=0;
	head_f3:=0;
	head_b:=0;
	head_f:=0;
	head_b2:=0;
	head_f2:=0;
	side_r:=0;
	side_l:=0;
END_IF

IF extend_do THEN
(*超过危险角度停车*)
	IF angle_x>angle_x_offset+400 OR angle_x<angle_x_offset-400 OR angle_x>angle_danger02+100 OR angle_x<angle_danger01+100  THEN
		extend_do:=0;
	END_IF
(*倾斜角度判定,四个区域方向的偏移*)
	IF         		 (angle_x>=angle_x_offset+10 	AND angle_y<=angle_y_offset )OR (angle_x>=angle_x_offset 	AND angle_y<=angle_y_offset-10 )	THEN angle_dir:=1;(*右前高*)(*铭之光传感器*)
		ELSIF	(angle_x>=angle_x_offset+10	 AND angle_y>=angle_y_offset)OR (angle_x>=angle_x_offset	AND angle_y>=angle_y_offset+10)  	THEN angle_dir:=2;(*右后高*)
		ELSIF	(angle_x<=angle_x_offset-10 	AND angle_y<=angle_y_offset )OR (angle_x<=angle_x_offset 	AND angle_y<=angle_y_offset-10 )	THEN angle_dir:=3;(*左前高*)
		ELSIF	(angle_x<=angle_x_offset-10 	AND angle_y>=angle_y_offset)OR (angle_x<=angle_x_offset 	AND angle_y>=angle_y_offset+10)  	THEN angle_dir:=4;(*左后高*)
		ELSE    angle_dir:=0;
	END_IF

(*————————————————————————————自动支腿第二步————————————————————————————————————————*)
(*伸垂直支腿*)
	IF head_b2 OR head_f2 THEN
		v_touch_speed:=500;
	ELSE
		v_touch_speed:=500;
	END_IF


	IF extend_step=2 THEN
		tem2:=INT_TO_DINT(v_touch_time)*1000;
		ton1(in:=1,pt:=DINT_TO_TIME(tem2));
		ton1();
		IF NOT front_right_urt_ex_check 		THEN right_front_desired	:=v_touch_speed; 	ELSE right_front_desired:=0; 	END_IF
		IF NOT front_left_urt_ex_check 		THEN left_front_desired		:=v_touch_speed; 	ELSE left_front_desired:=0; 		END_IF
		IF NOT back_right_urt_ex_check 	THEN right_back_desired	:=v_touch_speed; 	ELSE right_back_desired:=0; 	END_IF
		IF NOT back_left_urt_ex_check 		THEN left_back_desired		:=v_touch_speed; 	ELSE left_back_desired:=0; 		END_IF


(***********************sl**增加*****************************************start*)
(*
		tona1(in:=1,pt:=t#9s);
*)

		tona1(in:=1,pt:=leg_time);

	IF(tona1.Q)AND(NOT side_l) AND(NOT side_r)THEN
(***1***)

		IF NOT front_left_urt_ex_check1 AND NOT front_right_urt_ex_check1 AND NOT back_left_urt_ex_check1 AND NOT back_right_urt_ex_check1 THEN
			IF(head_b3)THEN
				IF NOT front_left_urt_ex_check1 		THEN left_front_desired		:=v_touch_speed; 	ELSE left_front_desired:=0; 		END_IF
				IF NOT front_right_urt_ex_check1 	THEN right_front_desired	:=v_touch_speed; 	ELSE right_front_desired:=0; 	END_IF
				IF NOT back_left_urt_ex_check1 		THEN left_back_desired		:=v_touch_speed; 	ELSE left_back_desired:=0; 		END_IF
				IF NOT back_right_urt_ex_check1 	THEN right_back_desired	:=v_touch_speed; 	ELSE right_back_desired:=0; 	END_IF
			END_IF
			IF(head_f3)THEN
				IF NOT front_left_urt_ex_check1 		THEN left_front_desired		:=v_touch_speed; 	ELSE left_front_desired:=0; 		END_IF
				IF NOT front_right_urt_ex_check1 	THEN right_front_desired	:=v_touch_speed; 	ELSE right_front_desired:=0; 	END_IF
				IF NOT back_left_urt_ex_check1 		THEN left_back_desired		:=v_touch_speed; 	ELSE left_back_desired:=0; 		END_IF
				IF NOT back_right_urt_ex_check1 	THEN right_back_desired	:=v_touch_speed; 	ELSE right_back_desired:=0; 	END_IF
			END_IF
			IF(head_b)THEN
				IF NOT front_left_urt_ex_check1 		THEN left_front_desired		:=v_touch_speed; 	ELSE left_front_desired:=0; 		END_IF
				IF NOT front_right_urt_ex_check1 	THEN right_front_desired	:=v_touch_speed; 	ELSE right_front_desired:=0; 	END_IF
				IF NOT back_left_urt_ex_check1 		THEN left_back_desired		:=v_touch_speed/2; 	ELSE left_back_desired:=0; 		END_IF
				IF NOT back_right_urt_ex_check1 	THEN right_back_desired	:=v_touch_speed/2; 	ELSE right_back_desired:=0; 	END_IF
			END_IF
			IF(head_f)THEN
				IF NOT front_left_urt_ex_check1 		THEN left_front_desired		:=v_touch_speed/2; 	ELSE left_front_desired:=0; 		END_IF
				IF NOT front_right_urt_ex_check1 	THEN right_front_desired	:=v_touch_speed/2; 	ELSE right_front_desired:=0; 	END_IF
				IF NOT back_left_urt_ex_check1 		THEN left_back_desired		:=v_touch_speed; 	ELSE left_back_desired:=0; 		END_IF
				IF NOT back_right_urt_ex_check1 	THEN right_back_desired	:=v_touch_speed; 	ELSE right_back_desired:=0; 	END_IF
			END_IF
			IF(head_b2)THEN
				IF NOT front_left_urt_ex_check1 		THEN left_front_desired		:=v_touch_speed; 	ELSE left_front_desired:=0; 		END_IF
				IF NOT front_right_urt_ex_check1 	THEN right_front_desired	:=v_touch_speed; 	ELSE right_front_desired:=0; 	END_IF
				IF NOT back_left_urt_ex_check1 		THEN left_back_desired		:=0					; 	ELSE left_back_desired:=0; 		END_IF
				IF NOT back_right_urt_ex_check1 	THEN right_back_desired	:=0					; 	ELSE right_back_desired:=0; 	END_IF
(*
				IF NOT back_left_urt_ex_check1 		THEN left_back_desired		:=v_touch_speed/3; 	ELSE left_back_desired:=0; 		END_IF
				IF NOT back_right_urt_ex_check1 	THEN right_back_desired	:=v_touch_speed/3; 	ELSE right_back_desired:=0; 	END_IF
*)
			END_IF
			IF(head_f2)THEN
(*
				IF NOT front_left_urt_ex_check1 		THEN left_front_desired		:=v_touch_speed/3; 	ELSE left_front_desired:=0; 		END_IF
				IF NOT front_right_urt_ex_check1 	THEN right_front_desired	:=v_touch_speed/3; 	ELSE right_front_desired:=0; 	END_IF
*)
				IF NOT front_left_urt_ex_check1 		THEN left_front_desired		:=0					; 	ELSE left_front_desired:=0; 		END_IF
				IF NOT front_right_urt_ex_check1 	THEN right_front_desired	:=0					; 	ELSE right_front_desired:=0; 	END_IF
				IF NOT back_left_urt_ex_check1 		THEN left_back_desired		:=v_touch_speed; 	ELSE left_back_desired:=0; 		END_IF
				IF NOT back_right_urt_ex_check1 	THEN right_back_desired	:=v_touch_speed; 	ELSE right_back_desired:=0; 	END_IF
			END_IF
		END_IF
(***4***)
			IF( front_left_urt_ex_check1 AND NOT front_right_urt_ex_check1 AND NOT back_left_urt_ex_check1 AND NOT back_right_urt_ex_check1)THEN
					left_front_desired		:=0;
					IF(head_b2)AND (angle_y-angle_y_offset>150)THEN
						IF NOT back_left_urt_ex_check1 		THEN left_back_desired		:=0;				 	ELSE left_back_desired:=0; 		END_IF
						IF NOT back_right_urt_ex_check1 	THEN right_back_desired	:=0;				 	ELSE right_back_desired:=0; 	END_IF
					END_IF
					IF(head_f2)AND (angle_y-angle_y_offset<-150)THEN
						IF NOT front_left_urt_ex_check1 		THEN left_front_desired		:=0;				 	ELSE left_front_desired:=0; 		END_IF
						IF NOT front_right_urt_ex_check1 	THEN right_front_desired	:=0;				 	ELSE right_front_desired:=0; 	END_IF
					END_IF
			END_IF
			IF( NOT front_left_urt_ex_check1 AND  front_right_urt_ex_check1 AND NOT back_left_urt_ex_check1 AND NOT back_right_urt_ex_check1)THEN
					right_front_desired	:=0;
					IF(head_b2)AND (angle_y-angle_y_offset>150)THEN
						IF NOT back_left_urt_ex_check1 		THEN left_back_desired		:=0;				 	ELSE left_back_desired:=0; 		END_IF
						IF NOT back_right_urt_ex_check1 	THEN right_back_desired	:=0;				 	ELSE right_back_desired:=0; 	END_IF
					END_IF
					IF(head_f2)AND (angle_y-angle_y_offset<-150)THEN
						IF NOT front_left_urt_ex_check1 		THEN left_front_desired		:=0;				 	ELSE left_front_desired:=0; 		END_IF
						IF NOT front_right_urt_ex_check1 	THEN right_front_desired	:=0;				 	ELSE right_front_desired:=0; 	END_IF
					END_IF
			END_IF
			IF( NOT front_left_urt_ex_check1 AND NOT front_right_urt_ex_check1 AND  back_left_urt_ex_check1 AND NOT back_right_urt_ex_check1)THEN
					left_back_desired		:=0;
					IF(head_b2)AND (angle_y-angle_y_offset>150)THEN
						IF NOT back_left_urt_ex_check1 		THEN left_back_desired		:=0;				 	ELSE left_back_desired:=0; 		END_IF
						IF NOT back_right_urt_ex_check1 	THEN right_back_desired	:=0;				 	ELSE right_back_desired:=0; 	END_IF
					END_IF
					IF(head_f2)AND (angle_y-angle_y_offset<-150)THEN
						IF NOT front_left_urt_ex_check1 		THEN left_front_desired		:=0;				 	ELSE left_front_desired:=0; 		END_IF
						IF NOT front_right_urt_ex_check1 	THEN right_front_desired	:=0;				 	ELSE right_front_desired:=0; 	END_IF
					END_IF
			END_IF
			IF( NOT front_left_urt_ex_check1 AND NOT front_right_urt_ex_check1 AND NOT back_left_urt_ex_check1 AND  back_right_urt_ex_check1)THEN
					right_back_desired	:=0;
					IF(head_b2)AND (angle_y-angle_y_offset>150)THEN
						IF NOT back_left_urt_ex_check1 		THEN left_back_desired		:=0;				 	ELSE left_back_desired:=0; 		END_IF
						IF NOT back_right_urt_ex_check1 	THEN right_back_desired	:=0;				 	ELSE right_back_desired:=0; 	END_IF
					END_IF
					IF(head_f2)AND (angle_y-angle_y_offset<-150)THEN
						IF NOT front_left_urt_ex_check1 		THEN left_front_desired		:=0;				 	ELSE left_front_desired:=0; 		END_IF
						IF NOT front_right_urt_ex_check1 	THEN right_front_desired	:=0;				 	ELSE right_front_desired:=0; 	END_IF
					END_IF
			END_IF
(***6***)

			IF( front_left_urt_ex_check1 AND front_right_urt_ex_check1 AND NOT back_left_urt_ex_check1 AND NOT back_right_urt_ex_check1)THEN
					IF(head_b3)THEN
						IF(angle_y-angle_y_offset>50)THEN
							left_front_desired		:=v_touch_speed;
							right_front_desired	:=v_touch_speed;
						ELSE
							left_front_desired		:=0;
							right_front_desired	:=0;
						END_IF
					END_IF
					IF(head_b2)AND (angle_y-angle_y_offset>150)THEN
						IF NOT back_left_urt_ex_check1 		THEN left_back_desired		:=0;				 	ELSE left_back_desired:=0; 		END_IF
						IF NOT back_right_urt_ex_check1 	THEN right_back_desired	:=0;				 	ELSE right_back_desired:=0; 	END_IF
					END_IF
					IF(head_f2)AND (angle_y-angle_y_offset<-150)THEN
						IF NOT front_left_urt_ex_check1 		THEN left_front_desired		:=0;				 	ELSE left_front_desired:=0; 		END_IF
						IF NOT front_right_urt_ex_check1 	THEN right_front_desired	:=0;				 	ELSE right_front_desired:=0; 	END_IF
					END_IF
(**djx_add_start**)
IF (angle_x-angle_x_offset>50) THEN right_front_desired:=0;END_IF
IF  (angle_x-angle_x_offset<-50) THEN left_front_desired:=0;END_IF
(**djx_add_end**)
			END_IF
			IF( NOT front_left_urt_ex_check1 AND NOT  front_right_urt_ex_check1 AND back_left_urt_ex_check1 AND  back_right_urt_ex_check1)THEN
					IF(head_f3)THEN
						IF(angle_y-angle_y_offset<-50)THEN
							left_back_desired		:=v_touch_speed;
							right_back_desired	:=v_touch_speed;
						ELSE
							left_back_desired		:=0;
							right_back_desired	:=0;
						END_IF
					END_IF
					IF(head_b2)AND (angle_y-angle_y_offset>150)THEN
						IF NOT back_left_urt_ex_check1 		THEN left_back_desired		:=0;				 	ELSE left_back_desired:=0; 		END_IF
						IF NOT back_right_urt_ex_check1 	THEN right_back_desired	:=0;				 	ELSE right_back_desired:=0; 	END_IF
					END_IF
					IF(head_f2)AND (angle_y-angle_y_offset<-150)THEN
						IF NOT front_left_urt_ex_check1 		THEN left_front_desired		:=0;				 	ELSE left_front_desired:=0; 		END_IF
						IF NOT front_right_urt_ex_check1 	THEN right_front_desired	:=0;				 	ELSE right_front_desired:=0; 	END_IF
					END_IF
(**djx_add_start**)
IF (angle_x-angle_x_offset>50) THEN right_back_desired:=0;END_IF
IF  (angle_x-angle_x_offset<-50) THEN left_back_desired:=0;END_IF
(**djx_add_end**)
			END_IF

			IF( front_left_urt_ex_check1 AND NOT front_right_urt_ex_check1 AND back_left_urt_ex_check1 AND NOT back_right_urt_ex_check1)THEN
					IF(head_b2)AND (angle_y-angle_y_offset>150)THEN
						IF NOT back_left_urt_ex_check1 		THEN left_back_desired		:=0;				 	ELSE left_back_desired:=0; 		END_IF
						IF NOT back_right_urt_ex_check1 	THEN right_back_desired	:=0;				 	ELSE right_back_desired:=0; 	END_IF
					END_IF
					IF(head_f2)AND (angle_y-angle_y_offset<-150)THEN
						IF NOT front_left_urt_ex_check1 		THEN left_front_desired		:=0;				 	ELSE left_front_desired:=0; 		END_IF
						IF NOT front_right_urt_ex_check1 	THEN right_front_desired	:=0;				 	ELSE right_front_desired:=0; 	END_IF
					END_IF

							left_front_desired		:=0;
							left_back_desired		:=0;
			END_IF
			IF( front_left_urt_ex_check1 AND NOT front_right_urt_ex_check1 AND NOT back_left_urt_ex_check1 AND back_right_urt_ex_check1)THEN
					IF(head_b2)AND (angle_y-angle_y_offset>150)THEN
						IF NOT back_left_urt_ex_check1 		THEN left_back_desired		:=0;				 	ELSE left_back_desired:=0; 		END_IF
						IF NOT back_right_urt_ex_check1 	THEN right_back_desired	:=0;				 	ELSE right_back_desired:=0; 	END_IF
					END_IF
					IF(head_f2)AND (angle_y-angle_y_offset<-150)THEN
						IF NOT front_left_urt_ex_check1 		THEN left_front_desired		:=0;				 	ELSE left_front_desired:=0; 		END_IF
						IF NOT front_right_urt_ex_check1 	THEN right_front_desired	:=0;				 	ELSE right_front_desired:=0; 	END_IF
					END_IF

							left_front_desired		:=0;
							right_back_desired	:=0;
			END_IF
			IF( NOT front_left_urt_ex_check1 AND front_right_urt_ex_check1 AND back_left_urt_ex_check1 AND NOT back_right_urt_ex_check1)THEN
					IF(head_b2)AND (angle_y-angle_y_offset>150)THEN
						IF NOT back_left_urt_ex_check1 		THEN left_back_desired		:=0;				 	ELSE left_back_desired:=0; 		END_IF
						IF NOT back_right_urt_ex_check1 	THEN right_back_desired	:=0;				 	ELSE right_back_desired:=0; 	END_IF
					END_IF
					IF(head_f2)AND (angle_y-angle_y_offset<-150)THEN
						IF NOT front_left_urt_ex_check1 		THEN left_front_desired		:=0;				 	ELSE left_front_desired:=0; 		END_IF
						IF NOT front_right_urt_ex_check1 	THEN right_front_desired	:=0;				 	ELSE right_front_desired:=0; 	END_IF
					END_IF

							right_front_desired	:=0;
							left_back_desired		:=0;
			END_IF
			IF( NOT front_left_urt_ex_check1 AND front_right_urt_ex_check1 AND NOT  back_left_urt_ex_check1 AND back_right_urt_ex_check1)THEN
					IF(head_b2)AND (angle_y-angle_y_offset>150)THEN
						IF NOT back_left_urt_ex_check1 		THEN left_back_desired		:=0;				 	ELSE left_back_desired:=0; 		END_IF
						IF NOT back_right_urt_ex_check1 	THEN right_back_desired	:=0;				 	ELSE right_back_desired:=0; 	END_IF
					END_IF
					IF(head_f2)AND (angle_y-angle_y_offset<-150)THEN
						IF NOT front_left_urt_ex_check1 		THEN left_front_desired		:=0;				 	ELSE left_front_desired:=0; 		END_IF
						IF NOT front_right_urt_ex_check1 	THEN right_front_desired	:=0;				 	ELSE right_front_desired:=0; 	END_IF
					END_IF

							right_front_desired	:=0;
							right_back_desired	:=0;
			END_IF

(***4***)
			IF( front_left_urt_ex_check1 AND front_right_urt_ex_check1 AND back_left_urt_ex_check1 AND NOT back_right_urt_ex_check1)THEN
					IF(head_b3)THEN
						IF(angle_y-angle_y_offset>50)THEN
							IF(angle_x-angle_x_offset>50)THEN
								left_front_desired		:=v_touch_speed;
								right_front_desired	:=v_touch_speed/2;
								left_back_desired		:=v_touch_speed/3;
							ELSE 	IF(angle_x-angle_x_offset<-50)THEN
								left_front_desired		:=v_touch_speed/2;
								right_front_desired	:=v_touch_speed;
								left_back_desired		:=0;
							ELSE
								left_front_desired		:=v_touch_speed;
								right_front_desired	:=v_touch_speed;
								left_back_desired		:=0;
							END_IF
							END_IF
						END_IF
					END_IF
			END_IF
			IF( front_left_urt_ex_check1 AND front_right_urt_ex_check1 AND NOT back_left_urt_ex_check1 AND back_right_urt_ex_check1)THEN
					IF(head_b3)THEN
						IF(angle_y-angle_y_offset>50)THEN
							IF(angle_x-angle_x_offset>50)THEN
								left_front_desired		:=v_touch_speed;
								right_front_desired	:=v_touch_speed/2;
								right_back_desired	:=0;
							ELSE 	IF(angle_x-angle_x_offset<-50)THEN
								left_front_desired		:=v_touch_speed/2;
								right_front_desired	:=v_touch_speed;
								right_back_desired	:=v_touch_speed/3;
							ELSE
								left_front_desired		:=v_touch_speed;
								right_front_desired	:=v_touch_speed;
								right_back_desired	:=0;
							END_IF
							END_IF
						END_IF
					END_IF
			END_IF
			IF( NOT front_left_urt_ex_check1 AND front_right_urt_ex_check1 AND  back_left_urt_ex_check1 AND back_right_urt_ex_check1)THEN
					IF(head_f3)THEN
						IF(angle_y-angle_y_offset<-50)THEN
							IF(angle_x-angle_x_offset>50)THEN
								left_back_desired		:=v_touch_speed;
								right_back_desired	:=v_touch_speed/2;
								right_front_desired	:=0;
							ELSE 	IF(angle_x-angle_x_offset<-50)THEN
								left_back_desired		:=v_touch_speed/2;
								right_back_desired	:=v_touch_speed;
								right_front_desired	:=v_touch_speed/3;
							ELSE
								left_back_desired		:=v_touch_speed;
								right_back_desired	:=v_touch_speed;
								right_front_desired	:=0;
							END_IF
							END_IF
						END_IF
					END_IF
			END_IF
			IF( front_left_urt_ex_check1 AND NOT front_right_urt_ex_check1 AND  back_left_urt_ex_check1 AND back_right_urt_ex_check1)THEN
					IF(head_f3)THEN
						IF(angle_y-angle_y_offset<-50)THEN
							IF(angle_x-angle_x_offset>50)THEN
								left_back_desired		:=v_touch_speed;
								right_back_desired	:=v_touch_speed/2;
								left_front_desired		:=v_touch_speed/3;
							ELSE 	IF(angle_x-angle_x_offset<-50)THEN
								left_back_desired		:=v_touch_speed/2;
								right_back_desired	:=v_touch_speed;
								left_front_desired		:=0;
							ELSE
								left_back_desired		:=v_touch_speed;
								right_back_desired	:=v_touch_speed;
								left_front_desired		:=0;
							END_IF
							END_IF
						END_IF
					END_IF
			END_IF


(***1***)

			IF( front_left_urt_ex_check1 AND  front_right_urt_ex_check1 AND  back_left_urt_ex_check1 AND back_right_urt_ex_check1)THEN
					IF(head_b3)THEN
						IF(angle_y-angle_y_offset>30)THEN
							IF(angle_x-angle_x_offset>50)THEN
								left_front_desired		:=v_touch_speed;
								right_front_desired	:=v_touch_speed/2;
								left_back_desired		:=v_touch_speed/3;
								right_back_desired	:=0;
							ELSE 	IF(angle_x-angle_x_offset<-50)THEN
								left_front_desired		:=v_touch_speed/2;
								right_front_desired	:=v_touch_speed;
								left_back_desired		:=0;
								right_back_desired	:=v_touch_speed/3;
							ELSE
								left_front_desired		:=v_touch_speed;
								right_front_desired	:=v_touch_speed;
								left_back_desired		:=0;
								right_back_desired	:=0;
							END_IF
							END_IF

						ELSE
							IF(angle_x-angle_x_offset>50)THEN
								left_front_desired		:=v_touch_speed/2;
								right_front_desired	:=0;
								left_back_desired		:=v_touch_speed/2;
								right_back_desired	:=0;
							ELSE 	IF(angle_x-angle_x_offset<-50)THEN
								left_front_desired		:=0;
								right_front_desired	:=v_touch_speed/2;
								left_back_desired		:=0;
								right_back_desired	:=v_touch_speed/2;
							END_IF
							END_IF
						END_IF
					END_IF
					IF(head_f3)THEN
						IF(angle_y-angle_y_offset<-30)THEN
							IF(angle_x-angle_x_offset>50)THEN
								left_front_desired		:=v_touch_speed/3;
								right_front_desired	:=0;
								left_back_desired		:=v_touch_speed;
								right_back_desired	:=v_touch_speed/2;
							ELSE 	IF(angle_x-angle_x_offset<-50)THEN
								left_front_desired		:=0;
								right_front_desired	:=v_touch_speed/3;
								left_back_desired		:=v_touch_speed/2;
								right_back_desired	:=v_touch_speed;
							ELSE
								left_front_desired		:=0;
								right_front_desired	:=0;
								left_back_desired		:=v_touch_speed;
								right_back_desired	:=v_touch_speed;

							END_IF
							END_IF

						ELSE
							IF(angle_x-angle_x_offset>50)THEN
								left_front_desired		:=v_touch_speed/2;
								right_front_desired	:=0;
								left_back_desired		:=v_touch_speed/2;
								right_back_desired	:=0;
							ELSE 	IF(angle_x-angle_x_offset<-50)THEN
								left_front_desired		:=0;
								right_front_desired	:=v_touch_speed/2;
								left_back_desired		:=0;
								right_back_desired	:=v_touch_speed/2;
							END_IF
							END_IF
						END_IF
					END_IF
				IF(((head_b3)AND(angle_y-angle_y_offset<=30))OR ((head_f3)AND(angle_y-angle_y_offset>=-30)))AND ABS(angle_x-angle_x_offset<=50)THEN
					step2_m2:=1;
				END_IF
			END_IF
		END_IF

		IF(side_r )THEN
			tona3(in:=1,pt:=t#9s);
			IF(tona3.Q AND tona_m3)THEN
				IF(front_left_urt_ex_check AND back_left_urt_ex_check)THEN
					 right_front_desired	:=0;
					 left_front_desired		:=v_touch_speed;
				 	right_back_desired	:=0;
				 	left_back_desired		:=v_touch_speed;
				END_IF
				IF(front_left_urt_ex_check AND NOT back_left_urt_ex_check)THEN   left_back_desired:=v_touch_speed; 	 left_front_desired	:=0; END_IF
				IF(NOT front_left_urt_ex_check AND  back_left_urt_ex_check)THEN   left_back_desired:=0; 	 left_front_desired	:=v_touch_speed;  END_IF
(*djx_add_start**********)
IF (angle_y-angle_y_offset>50)THEN left_back_desired:=0;END_IF
IF (angle_y-angle_y_offset<-50)THEN left_front_desired:=0;END_IF
(*djx_add_end*****************)
			END_IF
			IF(angle_x-angle_x_offset<50)THEN
				tona_m3:=0;
				IF(front_right_urt_ex_check AND back_right_urt_ex_check)THEN
					side_r:=0; side_m:=1;
				END_IF
			END_IF
		END_IF

		IF(side_l )THEN
			tona4(in:=1,pt:=t#9s);
			IF(tona4.Q AND tona_m4)THEN
				IF(front_right_urt_ex_check AND back_right_urt_ex_check)THEN
					 right_front_desired	:=v_touch_speed;
					 left_front_desired		:=0;
					 right_back_desired	:=v_touch_speed;
					 left_back_desired	:=0;
				END_IF
				IF(front_right_urt_ex_check AND NOT back_right_urt_ex_check)THEN   right_back_desired:=v_touch_speed; 	 right_front_desired	:=0;  END_IF
				IF(NOT front_right_urt_ex_check AND  back_right_urt_ex_check)THEN   right_back_desired:=0; 	right_front_desired:=v_touch_speed;  END_IF
(*djx_add_start**********)
IF (angle_y-angle_y_offset>50)THEN right_back_desired:=0;END_IF
IF (angle_y-angle_y_offset<-50)THEN right_front_desired:=0;END_IF
(*djx_add_end*****************)
			END_IF
			IF(angle_x-angle_x_offset>-50)THEN
				tona_m4:=0;
				IF(front_left_urt_ex_check AND back_left_urt_ex_check)THEN
					side_l:=0; side_m:=1;
				END_IF
			END_IF
		END_IF


(***********************sl**增加*******************************************end*)

		IF ((front_right_urt_ex_check AND front_left_urt_ex_check AND back_right_urt_ex_check AND back_left_urt_ex_check ) AND step2_m2)OR ton1.q THEN
			step2_m1:=0;
			step2_m2:=0;
			step2_m3:=0;
			step2_m4:=0;
			side_m:=0;
			ton1(in:=0);
(**增加部分-支腿二次调平***************)
			extend_step:=3;
			IF ((ABS(angle_x-angle_x_offset)<=100 AND( ((angle_y-angle_y_offset)>=-30 AND head_f3)OR((angle_y-angle_y_offset)<=30 AND head_b3)  ))OR (left_groud_check1 AND  left_groud_check2))	THEN
				(*IF(ABS(angle_x-angle_x_offset)<=angle_ok*2 AND three_step) OR ( left_groud_check1 AND  left_groud_check2)THEN*)
				extend_step:=4;
			ELSE extend_step:=3;
			END_IF
(*			IF (ABS(angle_x-angle_x_offset)<=150 AND ABS(angle_y-angle_y_offset)<=150)  THEN	extend_step:=4;ELSE extend_step:=3;END_IF*)
			fl_to_groud:=0;
			fr_to_groud:=0;
			bl_to_groud:=0;
			br_to_groud:=0;
			tona1(in:=0);
			tona2(in:=0);
			tona3(in:=0);
			tona4(in:=0);
		END_IF
	END_IF



(*————————————————————————————自动支腿第三步————————————————————————————————————————*)
(*粗调平过程，限时10s*)
	IF extend_step=3 THEN
		tona1(in:=0);
		tona2(in:=0);
		tona3(in:=0);
		tona4(in:=0);
		ton1(in:=1,pt:=t#10s);
		ton1();
		angle_x_real:=INT_TO_REAL(angle_x);
		angle_x_offset_real:=INT_TO_REAL(angle_x_offset);
		IF angle_x_real<angle_x_offset_real THEN
			PD1(ACTUAL:=angle_x_real ,SET_POINT:=angle_x_offset_real+50 , KP:=1 , TV:=1 , Y_MANUAL:=0 , 	Y_OFFSET:=0 , 	Y_MIN:=0 , 	Y_MAX:= 600,
			MANUAL:=FALSE , 	RESET:=FALSE , 	Y=>set_x_real , 	LIMITS_ACTIVE=>x_limit );
		ELSE
			PD2(ACTUAL:=angle_x_offset_real-angle_x_real ,SET_POINT:=50 , KP:=1 , TV:=1 , Y_MANUAL:=0 , 	Y_OFFSET:=0 , 	Y_MIN:=0 , 	Y_MAX:= 600,
			MANUAL:=FALSE , 	RESET:=FALSE , 	Y=>set_x_real , 	LIMITS_ACTIVE=>x_limit );
		END_IF
		set_x:=REAL_TO_WORD(ABS(set_x_real));

		angle_y_real:=INT_TO_REAL(angle_y);
		angle_y_offset_real:=INT_TO_REAL(angle_y_offset);
	IF(head_b3)THEN
		IF angle_y_real<angle_y_offset_real THEN
			PD3(ACTUAL:=angle_y_real ,SET_POINT:=angle_y_offset_real , KP:=1 , TV:=1 , Y_MANUAL:=0 , 	Y_OFFSET:=0 , 	Y_MIN:=0 , 	Y_MAX:= 600,
			MANUAL:=FALSE , 	RESET:=FALSE , 	Y=>set_y_real , 	LIMITS_ACTIVE=>y_limit );
		ELSE
			PD4(ACTUAL:=angle_y_offset_real-angle_y_real ,SET_POINT:=50 , KP:=1 , TV:=1 , Y_MANUAL:=0 , 	Y_OFFSET:=0 , 	Y_MIN:=0 , 	Y_MAX:= 600,
			MANUAL:=FALSE , 	RESET:=FALSE , 	Y=>set_y_real , 	LIMITS_ACTIVE=>y_limit );
		END_IF
		set_y:=REAL_TO_WORD(ABS(set_y_real));set_y := set_y*8/rl_ys;
	END_IF
	IF(head_f3)THEN
		IF angle_y_real<angle_y_offset_real THEN
			PD3(ACTUAL:=angle_y_real ,SET_POINT:=angle_y_offset_real+50 , KP:=1 , TV:=1 , Y_MANUAL:=0 , 	Y_OFFSET:=0 , 	Y_MIN:=0 , 	Y_MAX:= 600,
			MANUAL:=FALSE , 	RESET:=FALSE , 	Y=>set_y_real , 	LIMITS_ACTIVE=>y_limit );
		ELSE
			PD4(ACTUAL:=angle_y_offset_real-angle_y_real ,SET_POINT:=0 , KP:=1 , TV:=1 , Y_MANUAL:=0 , 	Y_OFFSET:=0 , 	Y_MIN:=0 , 	Y_MAX:= 600,
			MANUAL:=FALSE , 	RESET:=FALSE , 	Y=>set_y_real , 	LIMITS_ACTIVE=>y_limit );
		END_IF
		set_y:=REAL_TO_WORD(ABS(set_y_real));set_y := set_y*8/rl_ys;
	END_IF

(*不同倾斜角度的不同处理*)
			CASE angle_dir OF
				1:right_back_desired:=set_y;left_front_desired:=set_x;left_back_desired:=set_x+set_y;right_front_desired:=0;
				2:right_front_desired:=set_y;left_back_desired:=set_x;left_front_desired:=set_x+set_y;right_back_desired:=0;
				3:left_back_desired:=set_y;right_front_desired:=set_x;right_back_desired:=set_x+set_y;left_front_desired:=0;
				4:left_front_desired:=set_y;right_back_desired:=set_x;right_front_desired:=set_x+set_y;left_back_desired:=0;
			END_CASE;

					IF NOT back_left_urt_ex_check THEN
						left_back_desired:=left_back_desired*2;
						IF(left_back_desired=0)THEN left_back_desired:=right_back_desired*2;END_IF
						left_front_desired:=REAL_TO_WORD(WORD_TO_REAL(left_front_desired)/2);
						right_back_desired:=REAL_TO_WORD(WORD_TO_REAL(right_back_desired)/2);
					END_IF;
					IF NOT front_left_urt_ex_check THEN
						left_front_desired:=left_front_desired*2;
						IF(left_front_desired=0)THEN left_front_desired:=right_front_desired*2;END_IF
						left_back_desired:=REAL_TO_WORD(WORD_TO_REAL(left_back_desired)/2);
						right_front_desired:=REAL_TO_WORD(WORD_TO_REAL(right_front_desired)/2);
					END_IF;
					IF NOT back_right_urt_ex_check THEN
						right_back_desired:=right_back_desired*2;
						IF(right_back_desired=0)THEN right_back_desired:=left_back_desired*2;END_IF
						left_back_desired:=REAL_TO_WORD(WORD_TO_REAL(left_back_desired)/2);
						right_front_desired:=REAL_TO_WORD(WORD_TO_REAL(right_front_desired)/2);
					END_IF;
					IF NOT front_right_urt_ex_check THEN
						right_front_desired:=right_front_desired*2;
						IF(right_front_desired=0)THEN right_front_desired:=left_front_desired*2;END_IF
						left_front_desired:=REAL_TO_WORD(WORD_TO_REAL(left_front_desired)/2);
						right_back_desired:=REAL_TO_WORD(WORD_TO_REAL(right_back_desired)/2);
					END_IF;

		IF(head_b)THEN
			IF(angle_y-10<angle_y_offset)AND(angle_y-angle_y_offset>=-angle_ok*2)THEN three_step:=1; ELSE  three_step:=0; END_IF
		END_IF
		IF(head_f)THEN
			IF(angle_y+10>angle_y_offset)AND(angle_y-angle_y_offset<=angle_ok*2)THEN three_step:=1;  ELSE three_step:=0; END_IF
		END_IF
		IF(NOT head_b)AND(NOT head_f)OR(angle_dir=0)  THEN
			IF ABS(angle_y-angle_y_offset)<=angle_ok*2  THEN  three_step:=1; END_IF
		END_IF

		IF (ABS(angle_x-angle_x_offset)<=angle_ok*2 AND three_step) OR ( left_groud_check1 AND  left_groud_check2) OR ton1.q THEN
			ton1(in:=0);
			extend_step:=4;
			three_step:=0;
		END_IF
END_IF

(*————————————————————————————自动支腿第四步————————————————————————————————————————*)
(*撑起轮胎*)
	IF extend_step=4 THEN
		tem2:=INT_TO_DINT(v_rise_time)*1000;
		ton1(in:=1,pt:=DINT_TO_TIME(tem2));
		ton1();
		ton4_second(in:=level_second,pt:=t#3800ms);ton4_second();
		ton6_yanshi(in:=(NOT(left_groud_check1 AND left_groud_check2)),pt:=t#10000ms);ton6_yanshi();
		angle_x_real:=INT_TO_REAL(angle_x);
		angle_x_offset_real:=INT_TO_REAL(angle_x_offset);
		set_x:=REAL_TO_WORD(ABS(angle_x_real-angle_x_offset_real ));
		angle_y_real:=INT_TO_REAL(angle_y);
		angle_y_offset_real:=INT_TO_REAL(angle_y_offset);
		set_y:=REAL_TO_WORD(ABS(angle_y_real-angle_y_offset_real));set_y := set_y*8/rl_ys;
		IF ABS(angle_x-angle_x_offset)<step_4_limit AND ABS(angle_y-angle_y_offset)<step_4_limit THEN
			CASE angle_dir OF
				1:	left_front_desired:=REAL_TO_WORD(WORD_TO_REAL(v_rise_speed+set_x)*prop_m_1);
					right_back_desired:=REAL_TO_WORD(WORD_TO_REAL(v_rise_speed+set_y)*prop_m);
					left_back_desired:=REAL_TO_WORD(WORD_TO_REAL(v_rise_speed+set_y+set_x)*prop_m);
					right_front_desired:=REAL_TO_WORD(ABS(WORD_TO_REAL(v_rise_speed)-WORD_TO_REAL(set_y+set_x))*prop_m);
					IF left_back_desired<0 THEN left_back_desired:=1; END_IF
				2:	left_back_desired:=REAL_TO_WORD(WORD_TO_REAL(v_rise_speed+set_x)*prop_m);
					right_front_desired:=REAL_TO_WORD(WORD_TO_REAL(v_rise_speed+set_y)*prop_m);
					left_front_desired:=REAL_TO_WORD(WORD_TO_REAL(v_rise_speed+set_y+set_x)*prop_m_1);
					right_back_desired:=REAL_TO_WORD(ABS(WORD_TO_REAL(v_rise_speed)-WORD_TO_REAL(set_y+set_x))*prop_m);
					IF left_front_desired<0 THEN left_front_desired:=1; END_IF
				3:	right_front_desired:=REAL_TO_WORD(WORD_TO_REAL(v_rise_speed+set_x)*prop_m);
					left_back_desired:=REAL_TO_WORD(WORD_TO_REAL(v_rise_speed+set_y)*prop_m_1);
					right_back_desired:=REAL_TO_WORD(WORD_TO_REAL(v_rise_speed+set_y+set_x)*prop_m);
					left_front_desired:=REAL_TO_WORD(ABS(WORD_TO_REAL(v_rise_speed)-WORD_TO_REAL(set_y+set_x))*prop_m);
					IF right_back_desired<0 THEN right_back_desired:=1; END_IF
				4:	right_back_desired:=REAL_TO_WORD(WORD_TO_REAL(v_rise_speed+set_x)*prop_m);
					left_front_desired:=REAL_TO_WORD(WORD_TO_REAL(v_rise_speed+set_y)*prop_m);
					right_front_desired:=REAL_TO_WORD(WORD_TO_REAL(v_rise_speed+set_y+set_x)*prop_m);
					left_back_desired:=REAL_TO_WORD(ABS(WORD_TO_REAL(v_rise_speed)-WORD_TO_REAL(set_y+set_x))*prop_m);
					IF right_front_desired<0 THEN right_front_desired:=1; END_IF
			END_CASE

(*************sl 增加******************s*)
			IF(head_b AND (angle_y>angle_y_offset))THEN
				IF(angle_x>angle_x_offset)THEN
						left_front_desired:=left_front_desired+20;
						right_front_desired:=right_front_desired+15;
						left_back_desired:=left_back_desired-5;
						right_back_desired:=right_back_desired-10;
				END_IF
				IF(angle_x<angle_x_offset)THEN
						left_front_desired:=left_front_desired+15;
						right_front_desired:=right_front_desired+20;
						left_back_desired:=left_back_desired-10;
						right_back_desired:=right_back_desired-5;
				END_IF
			END_IF

			IF(head_b AND (angle_y<angle_y_offset))THEN
				IF(angle_x>angle_x_offset)THEN
						left_front_desired:=left_front_desired-5;
						right_front_desired:=right_front_desired-10;
						left_back_desired:=left_back_desired+15;
						right_back_desired:=right_back_desired+20;
				END_IF
				IF(angle_x<angle_x_offset)THEN
						left_front_desired:=left_front_desired-10;
						right_front_desired:=right_front_desired-5;
						left_back_desired:=left_back_desired+15;
						right_back_desired:=right_back_desired+20;
				END_IF
			END_IF

			IF(head_f AND (angle_y<angle_y_offset))THEN
				IF(angle_x>angle_x_offset)THEN
						left_front_desired:=left_front_desired-5;
						right_front_desired:=right_front_desired-10;
						left_back_desired:=left_back_desired+20;
						right_back_desired:=right_back_desired+15;
				END_IF
				IF(angle_x<angle_x_offset)THEN
						left_front_desired:=left_front_desired-10;
						right_front_desired:=right_front_desired-5;
						left_back_desired:=left_back_desired+15;
						right_back_desired:=right_back_desired+20;
				END_IF
			END_IF

			IF(head_f AND (angle_y>angle_y_offset))THEN
				IF(angle_x>angle_x_offset)THEN
						left_front_desired:=left_front_desired+20;
						right_front_desired:=right_front_desired+15;
						left_back_desired:=left_back_desired-5;
						right_back_desired:=right_back_desired-10;
				END_IF
				IF(angle_x<angle_x_offset)THEN
						left_front_desired:=left_front_desired+15;
						right_front_desired:=right_front_desired+20;
						left_back_desired:=left_back_desired-10;
						right_back_desired:=right_back_desired-5;
				END_IF
			END_IF

			IF(head_b AND (angle_y-30>angle_y_offset))THEN
				IF(angle_y_r1<angle_y_r2)THEN
					step4_m1:=step4_m1+1;
					step4_m2:=step4_m2+2;
					step4_m3:=0;
					step4_m4:=0;
				ELSE
					step4_m1:=0;
					step4_m2:=0;
				END_IF
				IF(angle_x>angle_x_offset)THEN
						left_front_desired:=left_front_desired+REAL_TO_WORD(step4_m2*1.0);
						right_front_desired:=right_front_desired+REAL_TO_WORD(step4_m2*0.6);
						left_back_desired:=left_back_desired-REAL_TO_WORD(step4_m1*0.5);
						right_back_desired:=right_back_desired-REAL_TO_WORD(step4_m1*1.0);
				END_IF
				IF(angle_x<angle_x_offset)THEN
						left_front_desired:=left_front_desired+REAL_TO_WORD(step4_m2*0.6);
						right_front_desired:=right_front_desired+REAL_TO_WORD(step4_m2*1.0);
						left_back_desired:=left_back_desired-REAL_TO_WORD(step4_m1*1.0);
						right_back_desired:=right_back_desired-REAL_TO_WORD(step4_m1*0.5);
				END_IF
			END_IF

			IF(head_f AND (angle_y+30<angle_y_offset))THEN
				IF(angle_y_r1>angle_y_r2)THEN
					step4_m1:=0;
					step4_m2:=0;
					step4_m3:=step4_m3+1;
					step4_m4:=step4_m4+2;
				ELSE
					step4_m3:=0;
					step4_m4:=0;
				END_IF
				IF(angle_x>angle_x_offset)THEN
						left_front_desired:=left_front_desired-REAL_TO_WORD(step4_m3*0.5);
						right_front_desired:=right_front_desired-REAL_TO_WORD(step4_m3*1.0);
						left_back_desired:=left_back_desired+REAL_TO_WORD(step4_m4*1.0);
						right_back_desired:=right_back_desired+REAL_TO_WORD(step4_m4*0.6);
				END_IF
				IF(angle_x<angle_x_offset)THEN
						left_front_desired:=left_front_desired-REAL_TO_WORD(step4_m3*1.0);
						right_front_desired:=right_front_desired-REAL_TO_WORD(step4_m3*0.5);
						left_back_desired:=left_back_desired+REAL_TO_WORD(step4_m4*0.6);
						right_back_desired:=right_back_desired+REAL_TO_WORD(step4_m4*1.0);
				END_IF
			END_IF


(*************sl 增加******************e*)

			IF NOT front_right_urt_ex_check1 THEN right_front_desired:=300; END_IF
			IF right_front_desired<0 THEN right_front_desired:=1; END_IF
			IF NOT front_left_urt_ex_check1 THEN left_front_desired:=300;END_IF
			IF left_front_desired<0 THEN left_front_desired:=1; END_IF
			IF NOT back_right_urt_ex_check1 THEN right_back_desired:=300; END_IF
			IF right_back_desired<0 THEN right_back_desired:=1; END_IF
			IF NOT back_left_urt_ex_check1 THEN left_back_desired:=300; END_IF
			IF left_back_desired<0 THEN left_back_desired:=1; END_IF
		END_IF
		IF ABS(angle_x-angle_x_offset)<step_4_limit AND (angle_y-angle_y_offset)<-step_4_limit THEN
			right_back_desired:=REAL_TO_WORD(WORD_TO_REAL(v_rise_speed)*prop_m);
			left_back_desired:=REAL_TO_WORD(WORD_TO_REAL(v_rise_speed)*prop_m_1);
		END_IF
		IF ABS(angle_x-angle_x_offset)<step_4_limit AND (angle_y-angle_y_offset)>step_4_limit THEN
			left_front_desired:=REAL_TO_WORD(WORD_TO_REAL(v_rise_speed)*prop_m);
			right_front_desired:=REAL_TO_WORD(WORD_TO_REAL(v_rise_speed)*prop_m_1);
		END_IF
		IF ABS(angle_y-angle_y_offset)<step_4_limit AND (angle_x-angle_x_offset)>step_4_limit THEN
			left_front_desired:=REAL_TO_WORD(WORD_TO_REAL(v_rise_speed)*prop_m);
			left_back_desired:=REAL_TO_WORD(WORD_TO_REAL(v_rise_speed)*prop_m_1);
		END_IF
		IF ABS(angle_y-angle_y_offset)<step_4_limit AND (angle_x-angle_x_offset)<-step_4_limit THEN
			right_back_desired:=REAL_TO_WORD(WORD_TO_REAL(v_rise_speed)*prop_m);
			right_front_desired:=REAL_TO_WORD(WORD_TO_REAL(v_rise_speed)*prop_m_1);
		END_IF

		IF ABS(angle_y-angle_y_offset)>step_4_limit AND ABS(angle_x-angle_x_offset)>step_4_limit THEN
			CASE angle_dir OF
				1:	left_front_desired:=REAL_TO_WORD(WORD_TO_REAL(v_rise_speed+set_x)*prop_m_1);
					right_back_desired:=REAL_TO_WORD(WORD_TO_REAL(v_rise_speed+set_y)*prop_m);
					left_back_desired:=REAL_TO_WORD(WORD_TO_REAL(v_rise_speed+set_y+set_x)*prop_m);
				2:	left_back_desired:=REAL_TO_WORD(WORD_TO_REAL(v_rise_speed+set_x)*prop_m);
					right_front_desired:=REAL_TO_WORD(WORD_TO_REAL(v_rise_speed+set_y)*prop_m);
					left_front_desired:=REAL_TO_WORD(WORD_TO_REAL(v_rise_speed+set_y+set_x)*prop_m_1);
				3:	right_front_desired:=REAL_TO_WORD(WORD_TO_REAL(v_rise_speed+set_x)*prop_m);
					left_back_desired:=REAL_TO_WORD(WORD_TO_REAL(v_rise_speed+set_y)*prop_m_1);
					right_back_desired:=REAL_TO_WORD(WORD_TO_REAL(v_rise_speed+set_y+set_x)*prop_m);
				4:	right_back_desired:=REAL_TO_WORD(WORD_TO_REAL(v_rise_speed+set_x)*prop_m);
					left_front_desired:=REAL_TO_WORD(WORD_TO_REAL(v_rise_speed+set_y)*prop_m);
					right_front_desired:=REAL_TO_WORD(WORD_TO_REAL(v_rise_speed+set_y+set_x)*prop_m);
			END_CASE
		END_IF
IF(left_front_desired<50)THEN left_front_desired:=50; END_IF
IF(right_back_desired<50)THEN right_back_desired:=50; END_IF
IF(right_front_desired<50)THEN right_front_desired:=50; END_IF
IF(left_back_desired<50)THEN left_back_desired:=50; END_IF

	IF (angle_y-angle_y_offset)<-step_4_limit+100 THEN left_front_desired:=0;right_front_desired:=0;END_IF
	IF (angle_y-angle_y_offset)>step_4_limit-100 THEN right_back_desired:=0;left_back_desired:=0;END_IF
	IF (angle_x-angle_x_offset)<-step_4_limit+100 THEN left_front_desired:=0;left_back_desired:=0;END_IF
	IF (angle_x-angle_x_offset)>step_4_limit-100 THEN right_back_desired:=0;right_front_desired:=0;END_IF


